(* PLC project tni_train, Dassault Systèmes ControlBuild 2019 FD01 Beta 2 *)
(* stored: creationDateTime 2018-09-11T17:45:24-01:00 *)

CONFIGURATION tni_train
  VAR_GLOBAL
    cab1/keyCabEnabled2 AT 97 : BOOL := false;
    cab1/keyCabDisabled2 AT 98 : BOOL := false;
    cab1/enableOpeningRightC1 AT 102 : BOOL := false;
    cab1/enableOpeningLeftC1 AT 104 : BOOL := false;
    cab1/enableClosingRightC1 AT 103 : BOOL := false;
    cab1/enableClosingLeftC1 AT 101 : BOOL := false;
    cab1/cabEnabled AT 99 : BOOL := false;
    cab1/cabDisabled AT 100 : BOOL := false;
    cab1/cabIncoherence AT 96 : BOOL := false;
    cab1/key2position/keyCabEnabled AT 109 : BOOL := false;
    cab1/key2position/keyCabDisabled AT 110 : BOOL := true;
    cab1/key2position/button AT 114 : BOOL := false;
    cab1/key2position/_X_10 AT 115 : BOOL := true;
    cab1/key2position/_X_11 AT 116 : BOOL := false;
    cab1/service_side/rightServiceSide AT 111 : BOOL := false;
    cab1/service_side/leftServiceSide AT 112 : BOOL := true;
    cab1/service_side/button AT 119 : BOOL := false;
    cab1/service_side/_X_10 AT 120 : BOOL := true;
    cab1/service_side/_X_11 AT 121 : BOOL := false;
    cab1/closingPB/PB AT 113 : BOOL := false;
    cab1/closingPB/button AT 124 : BOOL := false;
    cab1/closingPB/_X_10 AT 125 : BOOL := true;
    cab1/closingPB/_X_11 AT 126 : BOOL := false;
    cab1/trainSpeed/speed AT 17 : REAL := 0.0;
    cab1/cabControlPart/keyCabEnabled AT 109 : BOOL := false;
    cab1/cabControlPart/keyCabDisabled AT 110 : BOOL := true;
    cab1/cabControlPart/rightServiceSide AT 111 : BOOL := false;
    cab1/cabControlPart/leftServiceSide AT 112 : BOOL := true;
    cab1/cabControlPart/pbDoorClosing AT 113 : BOOL := false;
    cab1/cabControlPart/speed AT 17 : REAL := 0.0;
    cab1/cabControlPart/keyCabEnabled2 AT 97 : BOOL := false;
    cab1/cabControlPart/keyCabDisabled2 AT 98 : BOOL := false;
    cab1/cabControlPart/enableOpeningRightC1 AT 102 : BOOL := false;
    cab1/cabControlPart/enableOpeningLeftC1 AT 104 : BOOL := false;
    cab1/cabControlPart/enableClosingRightC1 AT 103 : BOOL := false;
    cab1/cabControlPart/enableClosingLeftC1 AT 101 : BOOL := false;
    cab1/cabControlPart/cabEnabled AT 99 : BOOL := false;
    cab1/cabControlPart/cabDisabled AT 100 : BOOL := false;
    cab1/cabControlPart/cabIncoherence AT 96 : BOOL := false;
    cab1/cabControlPart/limitLowSpeed AT 18 : REAL := 6.0;
    cab2/keyCabEnabled2 AT 99 : BOOL := false;
    cab2/keyCabDisabled2 AT 100 : BOOL := false;
    cab2/enableOpeningRightC1 AT 106 : BOOL := false;
    cab2/enableOpeningLeftC1 AT 108 : BOOL := false;
    cab2/enableClosingRightC1 AT 107 : BOOL := false;
    cab2/enableClosingLeftC1 AT 105 : BOOL := false;
    cab2/cabEnabled AT 97 : BOOL := false;
    cab2/cabDisabled AT 98 : BOOL := false;
    cab2/cabIncoherence AT 95 : BOOL := false;
    cab2/key2position/keyCabEnabled AT 129 : BOOL := false;
    cab2/key2position/keyCabDisabled AT 130 : BOOL := true;
    cab2/key2position/button AT 134 : BOOL := false;
    cab2/key2position/_X_10 AT 135 : BOOL := true;
    cab2/key2position/_X_11 AT 136 : BOOL := false;
    cab2/service_side/rightServiceSide AT 131 : BOOL := false;
    cab2/service_side/leftServiceSide AT 132 : BOOL := true;
    cab2/service_side/button AT 139 : BOOL := false;
    cab2/service_side/_X_10 AT 140 : BOOL := true;
    cab2/service_side/_X_11 AT 141 : BOOL := false;
    cab2/closingPB/PB AT 133 : BOOL := false;
    cab2/closingPB/button AT 144 : BOOL := false;
    cab2/closingPB/_X_10 AT 145 : BOOL := true;
    cab2/closingPB/_X_11 AT 146 : BOOL := false;
    cab2/trainSpeed/speed AT 19 : REAL := 0.0;
    cab2/cabControlPart/keyCabEnabled AT 129 : BOOL := false;
    cab2/cabControlPart/keyCabDisabled AT 130 : BOOL := true;
    cab2/cabControlPart/rightServiceSide AT 131 : BOOL := false;
    cab2/cabControlPart/leftServiceSide AT 132 : BOOL := true;
    cab2/cabControlPart/pbDoorClosing AT 133 : BOOL := false;
    cab2/cabControlPart/speed AT 19 : REAL := 0.0;
    cab2/cabControlPart/keyCabEnabled2 AT 99 : BOOL := false;
    cab2/cabControlPart/keyCabDisabled2 AT 100 : BOOL := false;
    cab2/cabControlPart/enableOpeningRightC1 AT 106 : BOOL := false;
    cab2/cabControlPart/enableOpeningLeftC1 AT 108 : BOOL := false;
    cab2/cabControlPart/enableClosingRightC1 AT 107 : BOOL := false;
    cab2/cabControlPart/enableClosingLeftC1 AT 105 : BOOL := false;
    cab2/cabControlPart/cabEnabled AT 97 : BOOL := false;
    cab2/cabControlPart/cabDisabled AT 98 : BOOL := false;
    cab2/cabControlPart/cabIncoherence AT 95 : BOOL := false;
    cab2/cabControlPart/limitLowSpeed AT 20 : REAL := 6.0;
    motorCar1/AuthorizationClosingLeftC1 AT 101 : BOOL := false;
    motorCar1/AuthorizationOpeningRightC1 AT 102 : BOOL := false;
    motorCar1/AuthorizationClosingRightC1 AT 103 : BOOL := false;
    motorCar1/AuthorizationOpeningLeftC1 AT 104 : BOOL := false;
    motorCar1/AuthorizationClosingLeftC2 AT 105 : BOOL := false;
    motorCar1/AuthorizationOpeningRightC2 AT 106 : BOOL := false;
    motorCar1/AuthorizationClosingRightC2 AT 107 : BOOL := false;
    motorCar1/AuthorizationOpeningLeftC2 AT 108 : BOOL := false;
    motorCar1/doorL1Closed AT 94 : BOOL := false;
    motorCar1/doorL1Opened AT 93 : BOOL := false;
    motorCar1/doorL1Fault AT 552 : DINT := 0;
    motorCar1/doorL2Closed AT 92 : BOOL := false;
    motorCar1/doorL2Opened AT 91 : BOOL := false;
    motorCar1/doorL2Fault AT 551 : DINT := 0;
    motorCar1/doorL3Closed AT 90 : BOOL := false;
    motorCar1/doorL3Opened AT 89 : BOOL := false;
    motorCar1/doorL3Fault AT 550 : DINT := 0;
    motorCar1/doorR1Closed AT 88 : BOOL := false;
    motorCar1/doorR1Opened AT 87 : BOOL := false;
    motorCar1/doorR1Fault AT 549 : DINT := 0;
    motorCar1/doorR2Closed AT 86 : BOOL := false;
    motorCar1/doorR2Opened AT 85 : BOOL := false;
    motorCar1/doorR2Fault AT 548 : DINT := 0;
    motorCar1/doorR3Closed AT 84 : BOOL := false;
    motorCar1/doorR3Opened AT 83 : BOOL := false;
    motorCar1/doorR3Fault AT 547 : DINT := 0;
    motorCar1/AlarmD1L AT 82 : BOOL := false;
    motorCar1/AlarmD2L AT 81 : BOOL := false;
    motorCar1/AlarmD3L AT 80 : BOOL := false;
    motorCar1/AlarmD1R AT 79 : BOOL := false;
    motorCar1/AlarmD2R AT 78 : BOOL := false;
    motorCar1/AlarmD3R AT 77 : BOOL := false;
    motorCar1/authorizations/AuthorizationClosingLeftC1 AT 101 : BOOL := false;
    motorCar1/authorizations/AuthorizationOpeningRightC1 AT 102 : BOOL := false;
    motorCar1/authorizations/AuthorizationClosingRightC1 AT 103 : BOOL := false;
    motorCar1/authorizations/AuthorizationOpeningLeftC1 AT 104 : BOOL := false;
    motorCar1/authorizations/AuthorizationClosingLeftC2 AT 105 : BOOL := false;
    motorCar1/authorizations/AuthorizationOpeningRightC2 AT 106 : BOOL := false;
    motorCar1/authorizations/AuthorizationClosingRightC2 AT 107 : BOOL := false;
    motorCar1/authorizations/AuthorizationOpeningLeftC2 AT 108 : BOOL := false;
    motorCar1/authorizations/AuthorizationOpeningLeft AT 161 : BOOL := false;
    motorCar1/authorizations/AuthorizationClosingLeft AT 162 : BOOL := false;
    motorCar1/authorizations/AuthorizationOpeningRight AT 163 : BOOL := false;
    motorCar1/authorizations/AuthorizationClosingRight AT 164 : BOOL := false;
    motorCar1/alarms/AlarmD1L AT 82 : BOOL := false;
    motorCar1/alarms/AlarmD2L AT 81 : BOOL := false;
    motorCar1/alarms/AlarmD3L AT 80 : BOOL := false;
    motorCar1/alarms/AlarmD1R AT 79 : BOOL := false;
    motorCar1/alarms/AlarmD2R AT 78 : BOOL := false;
    motorCar1/alarms/AlarmD3R AT 77 : BOOL := false;
    motorCar1/alarms/AlarmD1L/enableAlarm AT 176 : BOOL := false;
    motorCar1/alarms/AlarmD1L/resetKey AT 175 : BOOL := false;
    motorCar1/alarms/AlarmD1L/alarm AT 82 : BOOL := false;
    motorCar1/alarms/AlarmD1L/i_rs1 AT 553 : DINT := 0;
    motorCar1/alarms/AlarmD2L/enableAlarm AT 174 : BOOL := false;
    motorCar1/alarms/AlarmD2L/resetKey AT 173 : BOOL := false;
    motorCar1/alarms/AlarmD2L/alarm AT 81 : BOOL := false;
    motorCar1/alarms/AlarmD2L/i_rs1 AT 555 : DINT := 0;
    motorCar1/alarms/AlarmD3L/enableAlarm AT 172 : BOOL := false;
    motorCar1/alarms/AlarmD3L/resetKey AT 171 : BOOL := false;
    motorCar1/alarms/AlarmD3L/alarm AT 80 : BOOL := false;
    motorCar1/alarms/AlarmD3L/i_rs1 AT 557 : DINT := 0;
    motorCar1/alarms/AlarmD1R/enableAlarm AT 170 : BOOL := false;
    motorCar1/alarms/AlarmD1R/resetKey AT 169 : BOOL := false;
    motorCar1/alarms/AlarmD1R/alarm AT 79 : BOOL := false;
    motorCar1/alarms/AlarmD1R/i_rs1 AT 559 : DINT := 0;
    motorCar1/alarms/AlarmD2R/enableAlarm AT 168 : BOOL := false;
    motorCar1/alarms/AlarmD2R/resetKey AT 167 : BOOL := false;
    motorCar1/alarms/AlarmD2R/alarm AT 78 : BOOL := false;
    motorCar1/alarms/AlarmD2R/i_rs1 AT 561 : DINT := 0;
    motorCar1/alarms/AlarmD3R/enableAlarm AT 166 : BOOL := false;
    motorCar1/alarms/AlarmD3R/resetKey AT 165 : BOOL := false;
    motorCar1/alarms/AlarmD3R/alarm AT 77 : BOOL := false;
    motorCar1/alarms/AlarmD3R/i_rs1 AT 563 : DINT := 0;
    motorCar1/doorL1/compressedAir AT 26 : REAL := 200.0;
    motorCar1/doorL1/cmdSupply AT 160 : BOOL := true;
    motorCar1/doorL1/sensorSupply AT 159 : BOOL := true;
    motorCar1/doorL1/enableOpening AT 161 : BOOL := false;
    motorCar1/doorL1/enableClosing AT 162 : BOOL := false;
    motorCar1/doorL1/closedDoorState AT 94 : BOOL := false;
    motorCar1/doorL1/openedDoorState AT 93 : BOOL := false;
    motorCar1/doorL1/faultState AT 552 : DINT := 0;
    motorCar1/doorL1/doorPB/doorPB AT 189 : BOOL := false;
    motorCar1/doorL1/doorPB/button AT 193 : BOOL := false;
    motorCar1/doorL1/doorPB/_X_10 AT 194 : BOOL := true;
    motorCar1/doorL1/doorPB/_X_11 AT 195 : BOOL := false;
    motorCar1/doorL1/doorPB/_X_12 AT 196 : BOOL := false;
    motorCar1/doorL1/doorLocking/lockingCmd AT 183 : BOOL := false;
    motorCar1/doorL1/doorLocking/unlockingCmd AT 184 : BOOL := false;
    motorCar1/doorL1/doorLocking/doorLocked AT 187 : BOOL := false;
    motorCar1/doorL1/doorLocking/doorUnlocked AT 188 : BOOL := false;
    motorCar1/doorL1/doorLocking/lockActive AT 192 : BOOL := false;
    motorCar1/doorL1/doorLocking/i_rs1 AT 566 : DINT := 0;
    motorCar1/doorL1/doorLocking/d_unlockedSensor AT 198 : BOOL := false;
    motorCar1/doorL1/doorLocking/v_d_unlockedSensor AT 199 : BOOL := false;
    motorCar1/doorL1/doorLocking/d_lockedSensor AT 200 : BOOL := false;
    motorCar1/doorL1/doorLocking/v_d_lockedSensor AT 201 : BOOL := false;
    motorCar1/doorL1/doorControlPart/enableOpening AT 161 : BOOL := false;
    motorCar1/doorL1/doorControlPart/enableClosing AT 162 : BOOL := false;
    motorCar1/doorL1/doorControlPart/openedDoor AT 185 : BOOL := false;
    motorCar1/doorL1/doorControlPart/closedDoor AT 186 : BOOL := false;
    motorCar1/doorL1/doorControlPart/lockedDoor AT 187 : BOOL := false;
    motorCar1/doorL1/doorControlPart/unlockedDoor AT 188 : BOOL := false;
    motorCar1/doorL1/doorControlPart/openingRequest AT 189 : BOOL := false;
    motorCar1/doorL1/doorControlPart/doorOpeningCmd AT 190 : BOOL := false;
    motorCar1/doorL1/doorControlPart/doorClosingCmd AT 191 : BOOL := false;
    motorCar1/doorL1/doorControlPart/doorLockingCmd AT 183 : BOOL := false;
    motorCar1/doorL1/doorControlPart/doorUnlockingCmd AT 184 : BOOL := false;
    motorCar1/doorL1/doorControlPart/closedDoorState AT 94 : BOOL := false;
    motorCar1/doorL1/doorControlPart/openedDoorState AT 93 : BOOL := false;
    motorCar1/doorL1/doorControlPart/faultState AT 552 : DINT := 0;
    motorCar1/doorL1/doorControlPart/_X_10 AT 203 : BOOL := true;
    motorCar1/doorL1/doorControlPart/_X_11 AT 204 : BOOL := false;
    motorCar1/doorL1/doorControlPart/_X_12 AT 205 : BOOL := false;
    motorCar1/doorL1/doorControlPart/_X_13 AT 206 : BOOL := false;
    motorCar1/doorL1/doorControlPart/_X_14 AT 207 : BOOL := false;
    motorCar1/doorL1/doorControlPart/_X_15 AT 208 : BOOL := false;
    motorCar1/doorL1/doorControlPart/_X_16 AT 209 : BOOL := false;
    motorCar1/doorL1/door/compressedAir AT 26 : REAL := 200.0;
    motorCar1/doorL1/door/cmdSupply AT 160 : BOOL := true;
    motorCar1/doorL1/door/sensorSupply AT 159 : BOOL := true;
    motorCar1/doorL1/door/openDoorCmd AT 190 : BOOL := false;
    motorCar1/doorL1/door/closeDoorCmd AT 191 : BOOL := false;
    motorCar1/doorL1/door/lockActive AT 192 : BOOL := false;
    motorCar1/doorL1/door/doorOpened AT 185 : BOOL := false;
    motorCar1/doorL1/door/doorClosed AT 186 : BOOL := false;
    motorCar1/doorL1/door/increment AT 27 : REAL := 0.0;
    motorCar1/doorL1/door/openDoor AT 216 : BOOL := false;
    motorCar1/doorL1/door/closeDoor AT 217 : BOOL := false;
    motorCar1/doorL1/door/doorPosition AT 28 : REAL := 0.0;
    motorCar1/doorL1/door/length AT 29 : REAL := 1000.0;
    motorCar1/doorL1/door/doorClosedSensorLogic AT 218 : BOOL := true;
    motorCar1/doorL1/door/doorOpenedSensorLogic AT 219 : BOOL := true;
    motorCar1/doorL1/door/d_locking AT 220 : BOOL := false;
    motorCar1/doorL1/door/v_d_locking AT 30 : REAL := 50.0;
    motorCar1/doorL1/door/d_doorClosedSensor AT 221 : BOOL := false;
    motorCar1/doorL1/door/v_d_doorClosedSensor AT 222 : BOOL := false;
    motorCar1/doorL1/door/d_doorOpenedSensor AT 223 : BOOL := false;
    motorCar1/doorL1/door/v_d_doorOpenedSensor AT 224 : BOOL := false;
    motorCar1/doorL2/compressedAir AT 25 : REAL := 200.0;
    motorCar1/doorL2/cmdSupply AT 158 : BOOL := true;
    motorCar1/doorL2/sensorSupply AT 157 : BOOL := true;
    motorCar1/doorL2/enableOpening AT 161 : BOOL := false;
    motorCar1/doorL2/enableClosing AT 162 : BOOL := false;
    motorCar1/doorL2/closedDoorState AT 92 : BOOL := false;
    motorCar1/doorL2/openedDoorState AT 91 : BOOL := false;
    motorCar1/doorL2/faultState AT 551 : DINT := 0;
    motorCar1/doorL2/doorPB/doorPB AT 231 : BOOL := false;
    motorCar1/doorL2/doorPB/button AT 235 : BOOL := false;
    motorCar1/doorL2/doorPB/_X_10 AT 236 : BOOL := true;
    motorCar1/doorL2/doorPB/_X_11 AT 237 : BOOL := false;
    motorCar1/doorL2/doorPB/_X_12 AT 238 : BOOL := false;
    motorCar1/doorL2/doorLocking/lockingCmd AT 225 : BOOL := false;
    motorCar1/doorL2/doorLocking/unlockingCmd AT 226 : BOOL := false;
    motorCar1/doorL2/doorLocking/doorLocked AT 229 : BOOL := false;
    motorCar1/doorL2/doorLocking/doorUnlocked AT 230 : BOOL := false;
    motorCar1/doorL2/doorLocking/lockActive AT 234 : BOOL := false;
    motorCar1/doorL2/doorLocking/i_rs1 AT 569 : DINT := 0;
    motorCar1/doorL2/doorLocking/d_unlockedSensor AT 240 : BOOL := false;
    motorCar1/doorL2/doorLocking/v_d_unlockedSensor AT 241 : BOOL := false;
    motorCar1/doorL2/doorLocking/d_lockedSensor AT 242 : BOOL := false;
    motorCar1/doorL2/doorLocking/v_d_lockedSensor AT 243 : BOOL := false;
    motorCar1/doorL2/doorControlPart/enableOpening AT 161 : BOOL := false;
    motorCar1/doorL2/doorControlPart/enableClosing AT 162 : BOOL := false;
    motorCar1/doorL2/doorControlPart/openedDoor AT 227 : BOOL := false;
    motorCar1/doorL2/doorControlPart/closedDoor AT 228 : BOOL := false;
    motorCar1/doorL2/doorControlPart/lockedDoor AT 229 : BOOL := false;
    motorCar1/doorL2/doorControlPart/unlockedDoor AT 230 : BOOL := false;
    motorCar1/doorL2/doorControlPart/openingRequest AT 231 : BOOL := false;
    motorCar1/doorL2/doorControlPart/doorOpeningCmd AT 232 : BOOL := false;
    motorCar1/doorL2/doorControlPart/doorClosingCmd AT 233 : BOOL := false;
    motorCar1/doorL2/doorControlPart/doorLockingCmd AT 225 : BOOL := false;
    motorCar1/doorL2/doorControlPart/doorUnlockingCmd AT 226 : BOOL := false;
    motorCar1/doorL2/doorControlPart/closedDoorState AT 92 : BOOL := false;
    motorCar1/doorL2/doorControlPart/openedDoorState AT 91 : BOOL := false;
    motorCar1/doorL2/doorControlPart/faultState AT 551 : DINT := 0;
    motorCar1/doorL2/doorControlPart/_X_10 AT 245 : BOOL := true;
    motorCar1/doorL2/doorControlPart/_X_11 AT 246 : BOOL := false;
    motorCar1/doorL2/doorControlPart/_X_12 AT 247 : BOOL := false;
    motorCar1/doorL2/doorControlPart/_X_13 AT 248 : BOOL := false;
    motorCar1/doorL2/doorControlPart/_X_14 AT 249 : BOOL := false;
    motorCar1/doorL2/doorControlPart/_X_15 AT 250 : BOOL := false;
    motorCar1/doorL2/doorControlPart/_X_16 AT 251 : BOOL := false;
    motorCar1/doorL2/door/compressedAir AT 25 : REAL := 200.0;
    motorCar1/doorL2/door/cmdSupply AT 158 : BOOL := true;
    motorCar1/doorL2/door/sensorSupply AT 157 : BOOL := true;
    motorCar1/doorL2/door/openDoorCmd AT 232 : BOOL := false;
    motorCar1/doorL2/door/closeDoorCmd AT 233 : BOOL := false;
    motorCar1/doorL2/door/lockActive AT 234 : BOOL := false;
    motorCar1/doorL2/door/doorOpened AT 227 : BOOL := false;
    motorCar1/doorL2/door/doorClosed AT 228 : BOOL := false;
    motorCar1/doorL2/door/increment AT 31 : REAL := 0.0;
    motorCar1/doorL2/door/openDoor AT 258 : BOOL := false;
    motorCar1/doorL2/door/closeDoor AT 259 : BOOL := false;
    motorCar1/doorL2/door/doorPosition AT 32 : REAL := 0.0;
    motorCar1/doorL2/door/length AT 33 : REAL := 1000.0;
    motorCar1/doorL2/door/doorClosedSensorLogic AT 260 : BOOL := true;
    motorCar1/doorL2/door/doorOpenedSensorLogic AT 261 : BOOL := true;
    motorCar1/doorL2/door/d_locking AT 262 : BOOL := false;
    motorCar1/doorL2/door/v_d_locking AT 34 : REAL := 50.0;
    motorCar1/doorL2/door/d_doorClosedSensor AT 263 : BOOL := false;
    motorCar1/doorL2/door/v_d_doorClosedSensor AT 264 : BOOL := false;
    motorCar1/doorL2/door/d_doorOpenedSensor AT 265 : BOOL := false;
    motorCar1/doorL2/door/v_d_doorOpenedSensor AT 266 : BOOL := false;
    motorCar1/doorL3/compressedAir AT 24 : REAL := 200.0;
    motorCar1/doorL3/cmdSupply AT 156 : BOOL := true;
    motorCar1/doorL3/sensorSupply AT 155 : BOOL := true;
    motorCar1/doorL3/enableOpening AT 161 : BOOL := false;
    motorCar1/doorL3/enableClosing AT 162 : BOOL := false;
    motorCar1/doorL3/closedDoorState AT 90 : BOOL := false;
    motorCar1/doorL3/openedDoorState AT 89 : BOOL := false;
    motorCar1/doorL3/faultState AT 550 : DINT := 0;
    motorCar1/doorL3/doorPB/doorPB AT 273 : BOOL := false;
    motorCar1/doorL3/doorPB/button AT 277 : BOOL := false;
    motorCar1/doorL3/doorPB/_X_10 AT 278 : BOOL := true;
    motorCar1/doorL3/doorPB/_X_11 AT 279 : BOOL := false;
    motorCar1/doorL3/doorPB/_X_12 AT 280 : BOOL := false;
    motorCar1/doorL3/doorLocking/lockingCmd AT 267 : BOOL := false;
    motorCar1/doorL3/doorLocking/unlockingCmd AT 268 : BOOL := false;
    motorCar1/doorL3/doorLocking/doorLocked AT 271 : BOOL := false;
    motorCar1/doorL3/doorLocking/doorUnlocked AT 272 : BOOL := false;
    motorCar1/doorL3/doorLocking/lockActive AT 276 : BOOL := false;
    motorCar1/doorL3/doorLocking/i_rs1 AT 572 : DINT := 0;
    motorCar1/doorL3/doorLocking/d_unlockedSensor AT 282 : BOOL := false;
    motorCar1/doorL3/doorLocking/v_d_unlockedSensor AT 283 : BOOL := false;
    motorCar1/doorL3/doorLocking/d_lockedSensor AT 284 : BOOL := false;
    motorCar1/doorL3/doorLocking/v_d_lockedSensor AT 285 : BOOL := false;
    motorCar1/doorL3/doorControlPart/enableOpening AT 161 : BOOL := false;
    motorCar1/doorL3/doorControlPart/enableClosing AT 162 : BOOL := false;
    motorCar1/doorL3/doorControlPart/openedDoor AT 269 : BOOL := false;
    motorCar1/doorL3/doorControlPart/closedDoor AT 270 : BOOL := false;
    motorCar1/doorL3/doorControlPart/lockedDoor AT 271 : BOOL := false;
    motorCar1/doorL3/doorControlPart/unlockedDoor AT 272 : BOOL := false;
    motorCar1/doorL3/doorControlPart/openingRequest AT 273 : BOOL := false;
    motorCar1/doorL3/doorControlPart/doorOpeningCmd AT 274 : BOOL := false;
    motorCar1/doorL3/doorControlPart/doorClosingCmd AT 275 : BOOL := false;
    motorCar1/doorL3/doorControlPart/doorLockingCmd AT 267 : BOOL := false;
    motorCar1/doorL3/doorControlPart/doorUnlockingCmd AT 268 : BOOL := false;
    motorCar1/doorL3/doorControlPart/closedDoorState AT 90 : BOOL := false;
    motorCar1/doorL3/doorControlPart/openedDoorState AT 89 : BOOL := false;
    motorCar1/doorL3/doorControlPart/faultState AT 550 : DINT := 0;
    motorCar1/doorL3/doorControlPart/_X_10 AT 287 : BOOL := true;
    motorCar1/doorL3/doorControlPart/_X_11 AT 288 : BOOL := false;
    motorCar1/doorL3/doorControlPart/_X_12 AT 289 : BOOL := false;
    motorCar1/doorL3/doorControlPart/_X_13 AT 290 : BOOL := false;
    motorCar1/doorL3/doorControlPart/_X_14 AT 291 : BOOL := false;
    motorCar1/doorL3/doorControlPart/_X_15 AT 292 : BOOL := false;
    motorCar1/doorL3/doorControlPart/_X_16 AT 293 : BOOL := false;
    motorCar1/doorL3/door/compressedAir AT 24 : REAL := 200.0;
    motorCar1/doorL3/door/cmdSupply AT 156 : BOOL := true;
    motorCar1/doorL3/door/sensorSupply AT 155 : BOOL := true;
    motorCar1/doorL3/door/openDoorCmd AT 274 : BOOL := false;
    motorCar1/doorL3/door/closeDoorCmd AT 275 : BOOL := false;
    motorCar1/doorL3/door/lockActive AT 276 : BOOL := false;
    motorCar1/doorL3/door/doorOpened AT 269 : BOOL := false;
    motorCar1/doorL3/door/doorClosed AT 270 : BOOL := false;
    motorCar1/doorL3/door/increment AT 35 : REAL := 0.0;
    motorCar1/doorL3/door/openDoor AT 300 : BOOL := false;
    motorCar1/doorL3/door/closeDoor AT 301 : BOOL := false;
    motorCar1/doorL3/door/doorPosition AT 36 : REAL := 0.0;
    motorCar1/doorL3/door/length AT 37 : REAL := 1000.0;
    motorCar1/doorL3/door/doorClosedSensorLogic AT 302 : BOOL := true;
    motorCar1/doorL3/door/doorOpenedSensorLogic AT 303 : BOOL := true;
    motorCar1/doorL3/door/d_locking AT 304 : BOOL := false;
    motorCar1/doorL3/door/v_d_locking AT 38 : REAL := 50.0;
    motorCar1/doorL3/door/d_doorClosedSensor AT 305 : BOOL := false;
    motorCar1/doorL3/door/v_d_doorClosedSensor AT 306 : BOOL := false;
    motorCar1/doorL3/door/d_doorOpenedSensor AT 307 : BOOL := false;
    motorCar1/doorL3/door/v_d_doorOpenedSensor AT 308 : BOOL := false;
    motorCar1/doorR1/compressedAir AT 23 : REAL := 200.0;
    motorCar1/doorR1/cmdSupply AT 154 : BOOL := true;
    motorCar1/doorR1/sensorSupply AT 153 : BOOL := true;
    motorCar1/doorR1/enableOpening AT 163 : BOOL := false;
    motorCar1/doorR1/enableClosing AT 164 : BOOL := false;
    motorCar1/doorR1/closedDoorState AT 88 : BOOL := false;
    motorCar1/doorR1/openedDoorState AT 87 : BOOL := false;
    motorCar1/doorR1/faultState AT 549 : DINT := 0;
    motorCar1/doorR1/doorPB/doorPB AT 315 : BOOL := false;
    motorCar1/doorR1/doorPB/button AT 319 : BOOL := false;
    motorCar1/doorR1/doorPB/_X_10 AT 320 : BOOL := true;
    motorCar1/doorR1/doorPB/_X_11 AT 321 : BOOL := false;
    motorCar1/doorR1/doorPB/_X_12 AT 322 : BOOL := false;
    motorCar1/doorR1/doorLocking/lockingCmd AT 309 : BOOL := false;
    motorCar1/doorR1/doorLocking/unlockingCmd AT 310 : BOOL := false;
    motorCar1/doorR1/doorLocking/doorLocked AT 313 : BOOL := false;
    motorCar1/doorR1/doorLocking/doorUnlocked AT 314 : BOOL := false;
    motorCar1/doorR1/doorLocking/lockActive AT 318 : BOOL := false;
    motorCar1/doorR1/doorLocking/i_rs1 AT 575 : DINT := 0;
    motorCar1/doorR1/doorLocking/d_unlockedSensor AT 324 : BOOL := false;
    motorCar1/doorR1/doorLocking/v_d_unlockedSensor AT 325 : BOOL := false;
    motorCar1/doorR1/doorLocking/d_lockedSensor AT 326 : BOOL := false;
    motorCar1/doorR1/doorLocking/v_d_lockedSensor AT 327 : BOOL := false;
    motorCar1/doorR1/doorControlPart/enableOpening AT 163 : BOOL := false;
    motorCar1/doorR1/doorControlPart/enableClosing AT 164 : BOOL := false;
    motorCar1/doorR1/doorControlPart/openedDoor AT 311 : BOOL := false;
    motorCar1/doorR1/doorControlPart/closedDoor AT 312 : BOOL := false;
    motorCar1/doorR1/doorControlPart/lockedDoor AT 313 : BOOL := false;
    motorCar1/doorR1/doorControlPart/unlockedDoor AT 314 : BOOL := false;
    motorCar1/doorR1/doorControlPart/openingRequest AT 315 : BOOL := false;
    motorCar1/doorR1/doorControlPart/doorOpeningCmd AT 316 : BOOL := false;
    motorCar1/doorR1/doorControlPart/doorClosingCmd AT 317 : BOOL := false;
    motorCar1/doorR1/doorControlPart/doorLockingCmd AT 309 : BOOL := false;
    motorCar1/doorR1/doorControlPart/doorUnlockingCmd AT 310 : BOOL := false;
    motorCar1/doorR1/doorControlPart/closedDoorState AT 88 : BOOL := false;
    motorCar1/doorR1/doorControlPart/openedDoorState AT 87 : BOOL := false;
    motorCar1/doorR1/doorControlPart/faultState AT 549 : DINT := 0;
    motorCar1/doorR1/doorControlPart/_X_10 AT 329 : BOOL := true;
    motorCar1/doorR1/doorControlPart/_X_11 AT 330 : BOOL := false;
    motorCar1/doorR1/doorControlPart/_X_12 AT 331 : BOOL := false;
    motorCar1/doorR1/doorControlPart/_X_13 AT 332 : BOOL := false;
    motorCar1/doorR1/doorControlPart/_X_14 AT 333 : BOOL := false;
    motorCar1/doorR1/doorControlPart/_X_15 AT 334 : BOOL := false;
    motorCar1/doorR1/doorControlPart/_X_16 AT 335 : BOOL := false;
    motorCar1/doorR1/door/compressedAir AT 23 : REAL := 200.0;
    motorCar1/doorR1/door/cmdSupply AT 154 : BOOL := true;
    motorCar1/doorR1/door/sensorSupply AT 153 : BOOL := true;
    motorCar1/doorR1/door/openDoorCmd AT 316 : BOOL := false;
    motorCar1/doorR1/door/closeDoorCmd AT 317 : BOOL := false;
    motorCar1/doorR1/door/lockActive AT 318 : BOOL := false;
    motorCar1/doorR1/door/doorOpened AT 311 : BOOL := false;
    motorCar1/doorR1/door/doorClosed AT 312 : BOOL := false;
    motorCar1/doorR1/door/increment AT 39 : REAL := 0.0;
    motorCar1/doorR1/door/openDoor AT 342 : BOOL := false;
    motorCar1/doorR1/door/closeDoor AT 343 : BOOL := false;
    motorCar1/doorR1/door/doorPosition AT 40 : REAL := 0.0;
    motorCar1/doorR1/door/length AT 41 : REAL := 1000.0;
    motorCar1/doorR1/door/doorClosedSensorLogic AT 344 : BOOL := true;
    motorCar1/doorR1/door/doorOpenedSensorLogic AT 345 : BOOL := true;
    motorCar1/doorR1/door/d_locking AT 346 : BOOL := false;
    motorCar1/doorR1/door/v_d_locking AT 42 : REAL := 50.0;
    motorCar1/doorR1/door/d_doorClosedSensor AT 347 : BOOL := false;
    motorCar1/doorR1/door/v_d_doorClosedSensor AT 348 : BOOL := false;
    motorCar1/doorR1/door/d_doorOpenedSensor AT 349 : BOOL := false;
    motorCar1/doorR1/door/v_d_doorOpenedSensor AT 350 : BOOL := false;
    motorCar1/doorR2/compressedAir AT 22 : REAL := 200.0;
    motorCar1/doorR2/cmdSupply AT 152 : BOOL := true;
    motorCar1/doorR2/sensorSupply AT 151 : BOOL := true;
    motorCar1/doorR2/enableOpening AT 163 : BOOL := false;
    motorCar1/doorR2/enableClosing AT 164 : BOOL := false;
    motorCar1/doorR2/closedDoorState AT 86 : BOOL := false;
    motorCar1/doorR2/openedDoorState AT 85 : BOOL := false;
    motorCar1/doorR2/faultState AT 548 : DINT := 0;
    motorCar1/doorR2/doorPB/doorPB AT 357 : BOOL := false;
    motorCar1/doorR2/doorPB/button AT 361 : BOOL := false;
    motorCar1/doorR2/doorPB/_X_10 AT 362 : BOOL := true;
    motorCar1/doorR2/doorPB/_X_11 AT 363 : BOOL := false;
    motorCar1/doorR2/doorPB/_X_12 AT 364 : BOOL := false;
    motorCar1/doorR2/doorLocking/lockingCmd AT 351 : BOOL := false;
    motorCar1/doorR2/doorLocking/unlockingCmd AT 352 : BOOL := false;
    motorCar1/doorR2/doorLocking/doorLocked AT 355 : BOOL := false;
    motorCar1/doorR2/doorLocking/doorUnlocked AT 356 : BOOL := false;
    motorCar1/doorR2/doorLocking/lockActive AT 360 : BOOL := false;
    motorCar1/doorR2/doorLocking/i_rs1 AT 578 : DINT := 0;
    motorCar1/doorR2/doorLocking/d_unlockedSensor AT 366 : BOOL := false;
    motorCar1/doorR2/doorLocking/v_d_unlockedSensor AT 367 : BOOL := false;
    motorCar1/doorR2/doorLocking/d_lockedSensor AT 368 : BOOL := false;
    motorCar1/doorR2/doorLocking/v_d_lockedSensor AT 369 : BOOL := false;
    motorCar1/doorR2/doorControlPart/enableOpening AT 163 : BOOL := false;
    motorCar1/doorR2/doorControlPart/enableClosing AT 164 : BOOL := false;
    motorCar1/doorR2/doorControlPart/openedDoor AT 353 : BOOL := false;
    motorCar1/doorR2/doorControlPart/closedDoor AT 354 : BOOL := false;
    motorCar1/doorR2/doorControlPart/lockedDoor AT 355 : BOOL := false;
    motorCar1/doorR2/doorControlPart/unlockedDoor AT 356 : BOOL := false;
    motorCar1/doorR2/doorControlPart/openingRequest AT 357 : BOOL := false;
    motorCar1/doorR2/doorControlPart/doorOpeningCmd AT 358 : BOOL := false;
    motorCar1/doorR2/doorControlPart/doorClosingCmd AT 359 : BOOL := false;
    motorCar1/doorR2/doorControlPart/doorLockingCmd AT 351 : BOOL := false;
    motorCar1/doorR2/doorControlPart/doorUnlockingCmd AT 352 : BOOL := false;
    motorCar1/doorR2/doorControlPart/closedDoorState AT 86 : BOOL := false;
    motorCar1/doorR2/doorControlPart/openedDoorState AT 85 : BOOL := false;
    motorCar1/doorR2/doorControlPart/faultState AT 548 : DINT := 0;
    motorCar1/doorR2/doorControlPart/_X_10 AT 371 : BOOL := true;
    motorCar1/doorR2/doorControlPart/_X_11 AT 372 : BOOL := false;
    motorCar1/doorR2/doorControlPart/_X_12 AT 373 : BOOL := false;
    motorCar1/doorR2/doorControlPart/_X_13 AT 374 : BOOL := false;
    motorCar1/doorR2/doorControlPart/_X_14 AT 375 : BOOL := false;
    motorCar1/doorR2/doorControlPart/_X_15 AT 376 : BOOL := false;
    motorCar1/doorR2/doorControlPart/_X_16 AT 377 : BOOL := false;
    motorCar1/doorR2/door/compressedAir AT 22 : REAL := 200.0;
    motorCar1/doorR2/door/cmdSupply AT 152 : BOOL := true;
    motorCar1/doorR2/door/sensorSupply AT 151 : BOOL := true;
    motorCar1/doorR2/door/openDoorCmd AT 358 : BOOL := false;
    motorCar1/doorR2/door/closeDoorCmd AT 359 : BOOL := false;
    motorCar1/doorR2/door/lockActive AT 360 : BOOL := false;
    motorCar1/doorR2/door/doorOpened AT 353 : BOOL := false;
    motorCar1/doorR2/door/doorClosed AT 354 : BOOL := false;
    motorCar1/doorR2/door/increment AT 43 : REAL := 0.0;
    motorCar1/doorR2/door/openDoor AT 384 : BOOL := false;
    motorCar1/doorR2/door/closeDoor AT 385 : BOOL := false;
    motorCar1/doorR2/door/doorPosition AT 44 : REAL := 0.0;
    motorCar1/doorR2/door/length AT 45 : REAL := 1000.0;
    motorCar1/doorR2/door/doorClosedSensorLogic AT 386 : BOOL := true;
    motorCar1/doorR2/door/doorOpenedSensorLogic AT 387 : BOOL := true;
    motorCar1/doorR2/door/d_locking AT 388 : BOOL := false;
    motorCar1/doorR2/door/v_d_locking AT 46 : REAL := 50.0;
    motorCar1/doorR2/door/d_doorClosedSensor AT 389 : BOOL := false;
    motorCar1/doorR2/door/v_d_doorClosedSensor AT 390 : BOOL := false;
    motorCar1/doorR2/door/d_doorOpenedSensor AT 391 : BOOL := false;
    motorCar1/doorR2/door/v_d_doorOpenedSensor AT 392 : BOOL := false;
    motorCar1/doorR3/compressedAir AT 21 : REAL := 200.0;
    motorCar1/doorR3/cmdSupply AT 150 : BOOL := true;
    motorCar1/doorR3/sensorSupply AT 149 : BOOL := true;
    motorCar1/doorR3/enableOpening AT 163 : BOOL := false;
    motorCar1/doorR3/enableClosing AT 164 : BOOL := false;
    motorCar1/doorR3/closedDoorState AT 84 : BOOL := false;
    motorCar1/doorR3/openedDoorState AT 83 : BOOL := false;
    motorCar1/doorR3/faultState AT 547 : DINT := 0;
    motorCar1/doorR3/doorPB/doorPB AT 399 : BOOL := false;
    motorCar1/doorR3/doorPB/button AT 403 : BOOL := false;
    motorCar1/doorR3/doorPB/_X_10 AT 404 : BOOL := true;
    motorCar1/doorR3/doorPB/_X_11 AT 405 : BOOL := false;
    motorCar1/doorR3/doorPB/_X_12 AT 406 : BOOL := false;
    motorCar1/doorR3/doorLocking/lockingCmd AT 393 : BOOL := false;
    motorCar1/doorR3/doorLocking/unlockingCmd AT 394 : BOOL := false;
    motorCar1/doorR3/doorLocking/doorLocked AT 397 : BOOL := false;
    motorCar1/doorR3/doorLocking/doorUnlocked AT 398 : BOOL := false;
    motorCar1/doorR3/doorLocking/lockActive AT 402 : BOOL := false;
    motorCar1/doorR3/doorLocking/i_rs1 AT 581 : DINT := 0;
    motorCar1/doorR3/doorLocking/d_unlockedSensor AT 408 : BOOL := false;
    motorCar1/doorR3/doorLocking/v_d_unlockedSensor AT 409 : BOOL := false;
    motorCar1/doorR3/doorLocking/d_lockedSensor AT 410 : BOOL := false;
    motorCar1/doorR3/doorLocking/v_d_lockedSensor AT 411 : BOOL := false;
    motorCar1/doorR3/doorControlPart/enableOpening AT 163 : BOOL := false;
    motorCar1/doorR3/doorControlPart/enableClosing AT 164 : BOOL := false;
    motorCar1/doorR3/doorControlPart/openedDoor AT 395 : BOOL := false;
    motorCar1/doorR3/doorControlPart/closedDoor AT 396 : BOOL := false;
    motorCar1/doorR3/doorControlPart/lockedDoor AT 397 : BOOL := false;
    motorCar1/doorR3/doorControlPart/unlockedDoor AT 398 : BOOL := false;
    motorCar1/doorR3/doorControlPart/openingRequest AT 399 : BOOL := false;
    motorCar1/doorR3/doorControlPart/doorOpeningCmd AT 400 : BOOL := false;
    motorCar1/doorR3/doorControlPart/doorClosingCmd AT 401 : BOOL := false;
    motorCar1/doorR3/doorControlPart/doorLockingCmd AT 393 : BOOL := false;
    motorCar1/doorR3/doorControlPart/doorUnlockingCmd AT 394 : BOOL := false;
    motorCar1/doorR3/doorControlPart/closedDoorState AT 84 : BOOL := false;
    motorCar1/doorR3/doorControlPart/openedDoorState AT 83 : BOOL := false;
    motorCar1/doorR3/doorControlPart/faultState AT 547 : DINT := 0;
    motorCar1/doorR3/doorControlPart/_X_10 AT 413 : BOOL := true;
    motorCar1/doorR3/doorControlPart/_X_11 AT 414 : BOOL := false;
    motorCar1/doorR3/doorControlPart/_X_12 AT 415 : BOOL := false;
    motorCar1/doorR3/doorControlPart/_X_13 AT 416 : BOOL := false;
    motorCar1/doorR3/doorControlPart/_X_14 AT 417 : BOOL := false;
    motorCar1/doorR3/doorControlPart/_X_15 AT 418 : BOOL := false;
    motorCar1/doorR3/doorControlPart/_X_16 AT 419 : BOOL := false;
    motorCar1/doorR3/door/compressedAir AT 21 : REAL := 200.0;
    motorCar1/doorR3/door/cmdSupply AT 150 : BOOL := true;
    motorCar1/doorR3/door/sensorSupply AT 149 : BOOL := true;
    motorCar1/doorR3/door/openDoorCmd AT 400 : BOOL := false;
    motorCar1/doorR3/door/closeDoorCmd AT 401 : BOOL := false;
    motorCar1/doorR3/door/lockActive AT 402 : BOOL := false;
    motorCar1/doorR3/door/doorOpened AT 395 : BOOL := false;
    motorCar1/doorR3/door/doorClosed AT 396 : BOOL := false;
    motorCar1/doorR3/door/increment AT 47 : REAL := 0.0;
    motorCar1/doorR3/door/openDoor AT 426 : BOOL := false;
    motorCar1/doorR3/door/closeDoor AT 427 : BOOL := false;
    motorCar1/doorR3/door/doorPosition AT 48 : REAL := 0.0;
    motorCar1/doorR3/door/length AT 49 : REAL := 1000.0;
    motorCar1/doorR3/door/doorClosedSensorLogic AT 428 : BOOL := true;
    motorCar1/doorR3/door/doorOpenedSensorLogic AT 429 : BOOL := true;
    motorCar1/doorR3/door/d_locking AT 430 : BOOL := false;
    motorCar1/doorR3/door/v_d_locking AT 50 : REAL := 50.0;
    motorCar1/doorR3/door/d_doorClosedSensor AT 431 : BOOL := false;
    motorCar1/doorR3/door/v_d_doorClosedSensor AT 432 : BOOL := false;
    motorCar1/doorR3/door/d_doorOpenedSensor AT 433 : BOOL := false;
    motorCar1/doorR3/door/v_d_doorOpenedSensor AT 434 : BOOL := false;
    car1/AuthorizationClosingLeftC1 AT 101 : BOOL := false;
    car1/AuthorizationOpeningRightC1 AT 102 : BOOL := false;
    car1/AuthorizationClosingRightC1 AT 103 : BOOL := false;
    car1/AuthorizationOpeningLeftC1 AT 104 : BOOL := false;
    car1/AuthorizationClosingLeftC2 AT 105 : BOOL := false;
    car1/AuthorizationOpeningRightC2 AT 106 : BOOL := false;
    car1/AuthorizationClosingRightC2 AT 107 : BOOL := false;
    car1/AuthorizationOpeningLeftC2 AT 108 : BOOL := false;
    car1/doorL1Closed AT 76 : BOOL := false;
    car1/doorL1Opened AT 75 : BOOL := false;
    car1/doorL1Fault AT 546 : DINT := 0;
    car1/doorL2Closed AT 74 : BOOL := false;
    car1/doorL2Opened AT 73 : BOOL := false;
    car1/doorL2Fault AT 545 : DINT := 0;
    car1/doorL3Closed AT 72 : BOOL := false;
    car1/doorL3Opened AT 71 : BOOL := false;
    car1/doorL3Fault AT 544 : DINT := 0;
    car1/doorR1Closed AT 70 : BOOL := false;
    car1/doorR1Opened AT 69 : BOOL := false;
    car1/doorR1Fault AT 543 : DINT := 0;
    car1/doorR2Closed AT 68 : BOOL := false;
    car1/doorR2Opened AT 67 : BOOL := false;
    car1/doorR2Fault AT 542 : DINT := 0;
    car1/doorR3Closed AT 66 : BOOL := false;
    car1/doorR3Opened AT 65 : BOOL := false;
    car1/doorR3Fault AT 541 : DINT := 0;
    car1/AlarmD1L AT 64 : BOOL := false;
    car1/AlarmD2L AT 63 : BOOL := false;
    car1/AlarmD3L AT 62 : BOOL := false;
    car1/AlarmD1R AT 61 : BOOL := false;
    car1/AlarmD2R AT 60 : BOOL := false;
    car1/AlarmD3R AT 59 : BOOL := false;
    car1/authorizations/AuthorizationClosingLeftC1 AT 101 : BOOL := false;
    car1/authorizations/AuthorizationOpeningRightC1 AT 102 : BOOL := false;
    car1/authorizations/AuthorizationClosingRightC1 AT 103 : BOOL := false;
    car1/authorizations/AuthorizationOpeningLeftC1 AT 104 : BOOL := false;
    car1/authorizations/AuthorizationClosingLeftC2 AT 105 : BOOL := false;
    car1/authorizations/AuthorizationOpeningRightC2 AT 106 : BOOL := false;
    car1/authorizations/AuthorizationClosingRightC2 AT 107 : BOOL := false;
    car1/authorizations/AuthorizationOpeningLeftC2 AT 108 : BOOL := false;
    car1/authorizations/AuthorizationOpeningLeft AT 447 : BOOL := false;
    car1/authorizations/AuthorizationClosingLeft AT 448 : BOOL := false;
    car1/authorizations/AuthorizationOpeningRight AT 449 : BOOL := false;
    car1/authorizations/AuthorizationClosingRight AT 450 : BOOL := false;
    car1/alarms/AlarmD1L AT 64 : BOOL := false;
    car1/alarms/AlarmD2L AT 63 : BOOL := false;
    car1/alarms/AlarmD3L AT 62 : BOOL := false;
    car1/alarms/AlarmD1R AT 61 : BOOL := false;
    car1/alarms/AlarmD2R AT 60 : BOOL := false;
    car1/alarms/AlarmD3R AT 59 : BOOL := false;
    car1/alarms/AlarmD1L/enableAlarm AT 462 : BOOL := false;
    car1/alarms/AlarmD1L/resetKey AT 461 : BOOL := false;
    car1/alarms/AlarmD1L/alarm AT 64 : BOOL := false;
    car1/alarms/AlarmD1L/i_rs1 AT 583 : DINT := 0;
    car1/alarms/AlarmD2L/enableAlarm AT 460 : BOOL := false;
    car1/alarms/AlarmD2L/resetKey AT 459 : BOOL := false;
    car1/alarms/AlarmD2L/alarm AT 63 : BOOL := false;
    car1/alarms/AlarmD2L/i_rs1 AT 585 : DINT := 0;
    car1/alarms/AlarmD3L/enableAlarm AT 458 : BOOL := false;
    car1/alarms/AlarmD3L/resetKey AT 457 : BOOL := false;
    car1/alarms/AlarmD3L/alarm AT 62 : BOOL := false;
    car1/alarms/AlarmD3L/i_rs1 AT 587 : DINT := 0;
    car1/alarms/AlarmD1R/enableAlarm AT 456 : BOOL := false;
    car1/alarms/AlarmD1R/resetKey AT 455 : BOOL := false;
    car1/alarms/AlarmD1R/alarm AT 61 : BOOL := false;
    car1/alarms/AlarmD1R/i_rs1 AT 589 : DINT := 0;
    car1/alarms/AlarmD2R/enableAlarm AT 454 : BOOL := false;
    car1/alarms/AlarmD2R/resetKey AT 453 : BOOL := false;
    car1/alarms/AlarmD2R/alarm AT 60 : BOOL := false;
    car1/alarms/AlarmD2R/i_rs1 AT 591 : DINT := 0;
    car1/alarms/AlarmD3R/enableAlarm AT 452 : BOOL := false;
    car1/alarms/AlarmD3R/resetKey AT 451 : BOOL := false;
    car1/alarms/AlarmD3R/alarm AT 59 : BOOL := false;
    car1/alarms/AlarmD3R/i_rs1 AT 593 : DINT := 0;
    car1/doorL1/compressedAir AT 56 : REAL := 200.0;
    car1/doorL1/cmdSupply AT 446 : BOOL := true;
    car1/doorL1/sensorSupply AT 445 : BOOL := true;
    car1/doorL1/enableOpening AT 447 : BOOL := false;
    car1/doorL1/enableClosing AT 448 : BOOL := false;
    car1/doorL1/closedDoorState AT 76 : BOOL := false;
    car1/doorL1/openedDoorState AT 75 : BOOL := false;
    car1/doorL1/faultState AT 546 : DINT := 0;
    car1/doorL1/doorPB/doorPB AT 475 : BOOL := false;
    car1/doorL1/doorPB/button AT 479 : BOOL := false;
    car1/doorL1/doorPB/_X_10 AT 480 : BOOL := true;
    car1/doorL1/doorPB/_X_11 AT 481 : BOOL := false;
    car1/doorL1/doorPB/_X_12 AT 482 : BOOL := false;
    car1/doorL1/doorLocking/lockingCmd AT 469 : BOOL := false;
    car1/doorL1/doorLocking/unlockingCmd AT 470 : BOOL := false;
    car1/doorL1/doorLocking/doorLocked AT 473 : BOOL := false;
    car1/doorL1/doorLocking/doorUnlocked AT 474 : BOOL := false;
    car1/doorL1/doorLocking/lockActive AT 478 : BOOL := false;
    car1/doorL1/doorLocking/i_rs1 AT 596 : DINT := 0;
    car1/doorL1/doorLocking/d_unlockedSensor AT 484 : BOOL := false;
    car1/doorL1/doorLocking/v_d_unlockedSensor AT 485 : BOOL := false;
    car1/doorL1/doorLocking/d_lockedSensor AT 486 : BOOL := false;
    car1/doorL1/doorLocking/v_d_lockedSensor AT 487 : BOOL := false;
    car1/doorL1/doorControlPart/enableOpening AT 447 : BOOL := false;
    car1/doorL1/doorControlPart/enableClosing AT 448 : BOOL := false;
    car1/doorL1/doorControlPart/openedDoor AT 471 : BOOL := false;
    car1/doorL1/doorControlPart/closedDoor AT 472 : BOOL := false;
    car1/doorL1/doorControlPart/lockedDoor AT 473 : BOOL := false;
    car1/doorL1/doorControlPart/unlockedDoor AT 474 : BOOL := false;
    car1/doorL1/doorControlPart/openingRequest AT 475 : BOOL := false;
    car1/doorL1/doorControlPart/doorOpeningCmd AT 476 : BOOL := false;
    car1/doorL1/doorControlPart/doorClosingCmd AT 477 : BOOL := false;
    car1/doorL1/doorControlPart/doorLockingCmd AT 469 : BOOL := false;
    car1/doorL1/doorControlPart/doorUnlockingCmd AT 470 : BOOL := false;
    car1/doorL1/doorControlPart/closedDoorState AT 76 : BOOL := false;
    car1/doorL1/doorControlPart/openedDoorState AT 75 : BOOL := false;
    car1/doorL1/doorControlPart/faultState AT 546 : DINT := 0;
    car1/doorL1/doorControlPart/_X_10 AT 489 : BOOL := true;
    car1/doorL1/doorControlPart/_X_11 AT 490 : BOOL := false;
    car1/doorL1/doorControlPart/_X_12 AT 491 : BOOL := false;
    car1/doorL1/doorControlPart/_X_13 AT 492 : BOOL := false;
    car1/doorL1/doorControlPart/_X_14 AT 493 : BOOL := false;
    car1/doorL1/doorControlPart/_X_15 AT 494 : BOOL := false;
    car1/doorL1/doorControlPart/_X_16 AT 495 : BOOL := false;
    car1/doorL1/door/compressedAir AT 56 : REAL := 200.0;
    car1/doorL1/door/cmdSupply AT 446 : BOOL := true;
    car1/doorL1/door/sensorSupply AT 445 : BOOL := true;
    car1/doorL1/door/openDoorCmd AT 476 : BOOL := false;
    car1/doorL1/door/closeDoorCmd AT 477 : BOOL := false;
    car1/doorL1/door/lockActive AT 478 : BOOL := false;
    car1/doorL1/door/doorOpened AT 471 : BOOL := false;
    car1/doorL1/door/doorClosed AT 472 : BOOL := false;
    car1/doorL1/door/increment AT 57 : REAL := 0.0;
    car1/doorL1/door/openDoor AT 502 : BOOL := false;
    car1/doorL1/door/closeDoor AT 503 : BOOL := false;
    car1/doorL1/door/doorPosition AT 58 : REAL := 0.0;
    car1/doorL1/door/length AT 59 : REAL := 1000.0;
    car1/doorL1/door/doorClosedSensorLogic AT 504 : BOOL := true;
    car1/doorL1/door/doorOpenedSensorLogic AT 505 : BOOL := true;
    car1/doorL1/door/d_locking AT 506 : BOOL := false;
    car1/doorL1/door/v_d_locking AT 60 : REAL := 50.0;
    car1/doorL1/door/d_doorClosedSensor AT 507 : BOOL := false;
    car1/doorL1/door/v_d_doorClosedSensor AT 508 : BOOL := false;
    car1/doorL1/door/d_doorOpenedSensor AT 509 : BOOL := false;
    car1/doorL1/door/v_d_doorOpenedSensor AT 510 : BOOL := false;
    car1/doorL2/compressedAir AT 55 : REAL := 200.0;
    car1/doorL2/cmdSupply AT 444 : BOOL := true;
    car1/doorL2/sensorSupply AT 443 : BOOL := true;
    car1/doorL2/enableOpening AT 447 : BOOL := false;
    car1/doorL2/enableClosing AT 448 : BOOL := false;
    car1/doorL2/closedDoorState AT 74 : BOOL := false;
    car1/doorL2/openedDoorState AT 73 : BOOL := false;
    car1/doorL2/faultState AT 545 : DINT := 0;
    car1/doorL2/doorPB/doorPB AT 517 : BOOL := false;
    car1/doorL2/doorPB/button AT 521 : BOOL := false;
    car1/doorL2/doorPB/_X_10 AT 522 : BOOL := true;
    car1/doorL2/doorPB/_X_11 AT 523 : BOOL := false;
    car1/doorL2/doorPB/_X_12 AT 524 : BOOL := false;
    car1/doorL2/doorLocking/lockingCmd AT 511 : BOOL := false;
    car1/doorL2/doorLocking/unlockingCmd AT 512 : BOOL := false;
    car1/doorL2/doorLocking/doorLocked AT 515 : BOOL := false;
    car1/doorL2/doorLocking/doorUnlocked AT 516 : BOOL := false;
    car1/doorL2/doorLocking/lockActive AT 520 : BOOL := false;
    car1/doorL2/doorLocking/i_rs1 AT 599 : DINT := 0;
    car1/doorL2/doorLocking/d_unlockedSensor AT 526 : BOOL := false;
    car1/doorL2/doorLocking/v_d_unlockedSensor AT 527 : BOOL := false;
    car1/doorL2/doorLocking/d_lockedSensor AT 528 : BOOL := false;
    car1/doorL2/doorLocking/v_d_lockedSensor AT 529 : BOOL := false;
    car1/doorL2/doorControlPart/enableOpening AT 447 : BOOL := false;
    car1/doorL2/doorControlPart/enableClosing AT 448 : BOOL := false;
    car1/doorL2/doorControlPart/openedDoor AT 513 : BOOL := false;
    car1/doorL2/doorControlPart/closedDoor AT 514 : BOOL := false;
    car1/doorL2/doorControlPart/lockedDoor AT 515 : BOOL := false;
    car1/doorL2/doorControlPart/unlockedDoor AT 516 : BOOL := false;
    car1/doorL2/doorControlPart/openingRequest AT 517 : BOOL := false;
    car1/doorL2/doorControlPart/doorOpeningCmd AT 518 : BOOL := false;
    car1/doorL2/doorControlPart/doorClosingCmd AT 519 : BOOL := false;
    car1/doorL2/doorControlPart/doorLockingCmd AT 511 : BOOL := false;
    car1/doorL2/doorControlPart/doorUnlockingCmd AT 512 : BOOL := false;
    car1/doorL2/doorControlPart/closedDoorState AT 74 : BOOL := false;
    car1/doorL2/doorControlPart/openedDoorState AT 73 : BOOL := false;
    car1/doorL2/doorControlPart/faultState AT 545 : DINT := 0;
    car1/doorL2/doorControlPart/_X_10 AT 531 : BOOL := true;
    car1/doorL2/doorControlPart/_X_11 AT 532 : BOOL := false;
    car1/doorL2/doorControlPart/_X_12 AT 533 : BOOL := false;
    car1/doorL2/doorControlPart/_X_13 AT 534 : BOOL := false;
    car1/doorL2/doorControlPart/_X_14 AT 535 : BOOL := false;
    car1/doorL2/doorControlPart/_X_15 AT 536 : BOOL := false;
    car1/doorL2/doorControlPart/_X_16 AT 537 : BOOL := false;
    car1/doorL2/door/compressedAir AT 55 : REAL := 200.0;
    car1/doorL2/door/cmdSupply AT 444 : BOOL := true;
    car1/doorL2/door/sensorSupply AT 443 : BOOL := true;
    car1/doorL2/door/openDoorCmd AT 518 : BOOL := false;
    car1/doorL2/door/closeDoorCmd AT 519 : BOOL := false;
    car1/doorL2/door/lockActive AT 520 : BOOL := false;
    car1/doorL2/door/doorOpened AT 513 : BOOL := false;
    car1/doorL2/door/doorClosed AT 514 : BOOL := false;
    car1/doorL2/door/increment AT 61 : REAL := 0.0;
    car1/doorL2/door/openDoor AT 544 : BOOL := false;
    car1/doorL2/door/closeDoor AT 545 : BOOL := false;
    car1/doorL2/door/doorPosition AT 62 : REAL := 0.0;
    car1/doorL2/door/length AT 63 : REAL := 1000.0;
    car1/doorL2/door/doorClosedSensorLogic AT 546 : BOOL := true;
    car1/doorL2/door/doorOpenedSensorLogic AT 547 : BOOL := true;
    car1/doorL2/door/d_locking AT 548 : BOOL := false;
    car1/doorL2/door/v_d_locking AT 64 : REAL := 50.0;
    car1/doorL2/door/d_doorClosedSensor AT 549 : BOOL := false;
    car1/doorL2/door/v_d_doorClosedSensor AT 550 : BOOL := false;
    car1/doorL2/door/d_doorOpenedSensor AT 551 : BOOL := false;
    car1/doorL2/door/v_d_doorOpenedSensor AT 552 : BOOL := false;
    car1/doorL3/compressedAir AT 54 : REAL := 200.0;
    car1/doorL3/cmdSupply AT 442 : BOOL := true;
    car1/doorL3/sensorSupply AT 441 : BOOL := true;
    car1/doorL3/enableOpening AT 447 : BOOL := false;
    car1/doorL3/enableClosing AT 448 : BOOL := false;
    car1/doorL3/closedDoorState AT 72 : BOOL := false;
    car1/doorL3/openedDoorState AT 71 : BOOL := false;
    car1/doorL3/faultState AT 544 : DINT := 0;
    car1/doorL3/doorPB/doorPB AT 559 : BOOL := false;
    car1/doorL3/doorPB/button AT 563 : BOOL := false;
    car1/doorL3/doorPB/_X_10 AT 564 : BOOL := true;
    car1/doorL3/doorPB/_X_11 AT 565 : BOOL := false;
    car1/doorL3/doorPB/_X_12 AT 566 : BOOL := false;
    car1/doorL3/doorLocking/lockingCmd AT 553 : BOOL := false;
    car1/doorL3/doorLocking/unlockingCmd AT 554 : BOOL := false;
    car1/doorL3/doorLocking/doorLocked AT 557 : BOOL := false;
    car1/doorL3/doorLocking/doorUnlocked AT 558 : BOOL := false;
    car1/doorL3/doorLocking/lockActive AT 562 : BOOL := false;
    car1/doorL3/doorLocking/i_rs1 AT 602 : DINT := 0;
    car1/doorL3/doorLocking/d_unlockedSensor AT 568 : BOOL := false;
    car1/doorL3/doorLocking/v_d_unlockedSensor AT 569 : BOOL := false;
    car1/doorL3/doorLocking/d_lockedSensor AT 570 : BOOL := false;
    car1/doorL3/doorLocking/v_d_lockedSensor AT 571 : BOOL := false;
    car1/doorL3/doorControlPart/enableOpening AT 447 : BOOL := false;
    car1/doorL3/doorControlPart/enableClosing AT 448 : BOOL := false;
    car1/doorL3/doorControlPart/openedDoor AT 555 : BOOL := false;
    car1/doorL3/doorControlPart/closedDoor AT 556 : BOOL := false;
    car1/doorL3/doorControlPart/lockedDoor AT 557 : BOOL := false;
    car1/doorL3/doorControlPart/unlockedDoor AT 558 : BOOL := false;
    car1/doorL3/doorControlPart/openingRequest AT 559 : BOOL := false;
    car1/doorL3/doorControlPart/doorOpeningCmd AT 560 : BOOL := false;
    car1/doorL3/doorControlPart/doorClosingCmd AT 561 : BOOL := false;
    car1/doorL3/doorControlPart/doorLockingCmd AT 553 : BOOL := false;
    car1/doorL3/doorControlPart/doorUnlockingCmd AT 554 : BOOL := false;
    car1/doorL3/doorControlPart/closedDoorState AT 72 : BOOL := false;
    car1/doorL3/doorControlPart/openedDoorState AT 71 : BOOL := false;
    car1/doorL3/doorControlPart/faultState AT 544 : DINT := 0;
    car1/doorL3/doorControlPart/_X_10 AT 573 : BOOL := true;
    car1/doorL3/doorControlPart/_X_11 AT 574 : BOOL := false;
    car1/doorL3/doorControlPart/_X_12 AT 575 : BOOL := false;
    car1/doorL3/doorControlPart/_X_13 AT 576 : BOOL := false;
    car1/doorL3/doorControlPart/_X_14 AT 577 : BOOL := false;
    car1/doorL3/doorControlPart/_X_15 AT 578 : BOOL := false;
    car1/doorL3/doorControlPart/_X_16 AT 579 : BOOL := false;
    car1/doorL3/door/compressedAir AT 54 : REAL := 200.0;
    car1/doorL3/door/cmdSupply AT 442 : BOOL := true;
    car1/doorL3/door/sensorSupply AT 441 : BOOL := true;
    car1/doorL3/door/openDoorCmd AT 560 : BOOL := false;
    car1/doorL3/door/closeDoorCmd AT 561 : BOOL := false;
    car1/doorL3/door/lockActive AT 562 : BOOL := false;
    car1/doorL3/door/doorOpened AT 555 : BOOL := false;
    car1/doorL3/door/doorClosed AT 556 : BOOL := false;
    car1/doorL3/door/increment AT 65 : REAL := 0.0;
    car1/doorL3/door/openDoor AT 586 : BOOL := false;
    car1/doorL3/door/closeDoor AT 587 : BOOL := false;
    car1/doorL3/door/doorPosition AT 66 : REAL := 0.0;
    car1/doorL3/door/length AT 67 : REAL := 1000.0;
    car1/doorL3/door/doorClosedSensorLogic AT 588 : BOOL := true;
    car1/doorL3/door/doorOpenedSensorLogic AT 589 : BOOL := true;
    car1/doorL3/door/d_locking AT 590 : BOOL := false;
    car1/doorL3/door/v_d_locking AT 68 : REAL := 50.0;
    car1/doorL3/door/d_doorClosedSensor AT 591 : BOOL := false;
    car1/doorL3/door/v_d_doorClosedSensor AT 592 : BOOL := false;
    car1/doorL3/door/d_doorOpenedSensor AT 593 : BOOL := false;
    car1/doorL3/door/v_d_doorOpenedSensor AT 594 : BOOL := false;
    car1/doorR1/compressedAir AT 53 : REAL := 200.0;
    car1/doorR1/cmdSupply AT 440 : BOOL := true;
    car1/doorR1/sensorSupply AT 439 : BOOL := true;
    car1/doorR1/enableOpening AT 449 : BOOL := false;
    car1/doorR1/enableClosing AT 450 : BOOL := false;
    car1/doorR1/closedDoorState AT 70 : BOOL := false;
    car1/doorR1/openedDoorState AT 69 : BOOL := false;
    car1/doorR1/faultState AT 543 : DINT := 0;
    car1/doorR1/doorPB/doorPB AT 601 : BOOL := false;
    car1/doorR1/doorPB/button AT 605 : BOOL := false;
    car1/doorR1/doorPB/_X_10 AT 606 : BOOL := true;
    car1/doorR1/doorPB/_X_11 AT 607 : BOOL := false;
    car1/doorR1/doorPB/_X_12 AT 608 : BOOL := false;
    car1/doorR1/doorLocking/lockingCmd AT 595 : BOOL := false;
    car1/doorR1/doorLocking/unlockingCmd AT 596 : BOOL := false;
    car1/doorR1/doorLocking/doorLocked AT 599 : BOOL := false;
    car1/doorR1/doorLocking/doorUnlocked AT 600 : BOOL := false;
    car1/doorR1/doorLocking/lockActive AT 604 : BOOL := false;
    car1/doorR1/doorLocking/i_rs1 AT 605 : DINT := 0;
    car1/doorR1/doorLocking/d_unlockedSensor AT 610 : BOOL := false;
    car1/doorR1/doorLocking/v_d_unlockedSensor AT 611 : BOOL := false;
    car1/doorR1/doorLocking/d_lockedSensor AT 612 : BOOL := false;
    car1/doorR1/doorLocking/v_d_lockedSensor AT 613 : BOOL := false;
    car1/doorR1/doorControlPart/enableOpening AT 449 : BOOL := false;
    car1/doorR1/doorControlPart/enableClosing AT 450 : BOOL := false;
    car1/doorR1/doorControlPart/openedDoor AT 597 : BOOL := false;
    car1/doorR1/doorControlPart/closedDoor AT 598 : BOOL := false;
    car1/doorR1/doorControlPart/lockedDoor AT 599 : BOOL := false;
    car1/doorR1/doorControlPart/unlockedDoor AT 600 : BOOL := false;
    car1/doorR1/doorControlPart/openingRequest AT 601 : BOOL := false;
    car1/doorR1/doorControlPart/doorOpeningCmd AT 602 : BOOL := false;
    car1/doorR1/doorControlPart/doorClosingCmd AT 603 : BOOL := false;
    car1/doorR1/doorControlPart/doorLockingCmd AT 595 : BOOL := false;
    car1/doorR1/doorControlPart/doorUnlockingCmd AT 596 : BOOL := false;
    car1/doorR1/doorControlPart/closedDoorState AT 70 : BOOL := false;
    car1/doorR1/doorControlPart/openedDoorState AT 69 : BOOL := false;
    car1/doorR1/doorControlPart/faultState AT 543 : DINT := 0;
    car1/doorR1/doorControlPart/_X_10 AT 615 : BOOL := true;
    car1/doorR1/doorControlPart/_X_11 AT 616 : BOOL := false;
    car1/doorR1/doorControlPart/_X_12 AT 617 : BOOL := false;
    car1/doorR1/doorControlPart/_X_13 AT 618 : BOOL := false;
    car1/doorR1/doorControlPart/_X_14 AT 619 : BOOL := false;
    car1/doorR1/doorControlPart/_X_15 AT 620 : BOOL := false;
    car1/doorR1/doorControlPart/_X_16 AT 621 : BOOL := false;
    car1/doorR1/door/compressedAir AT 53 : REAL := 200.0;
    car1/doorR1/door/cmdSupply AT 440 : BOOL := true;
    car1/doorR1/door/sensorSupply AT 439 : BOOL := true;
    car1/doorR1/door/openDoorCmd AT 602 : BOOL := false;
    car1/doorR1/door/closeDoorCmd AT 603 : BOOL := false;
    car1/doorR1/door/lockActive AT 604 : BOOL := false;
    car1/doorR1/door/doorOpened AT 597 : BOOL := false;
    car1/doorR1/door/doorClosed AT 598 : BOOL := false;
    car1/doorR1/door/increment AT 69 : REAL := 0.0;
    car1/doorR1/door/openDoor AT 628 : BOOL := false;
    car1/doorR1/door/closeDoor AT 629 : BOOL := false;
    car1/doorR1/door/doorPosition AT 70 : REAL := 0.0;
    car1/doorR1/door/length AT 71 : REAL := 1000.0;
    car1/doorR1/door/doorClosedSensorLogic AT 630 : BOOL := true;
    car1/doorR1/door/doorOpenedSensorLogic AT 631 : BOOL := true;
    car1/doorR1/door/d_locking AT 632 : BOOL := false;
    car1/doorR1/door/v_d_locking AT 72 : REAL := 50.0;
    car1/doorR1/door/d_doorClosedSensor AT 633 : BOOL := false;
    car1/doorR1/door/v_d_doorClosedSensor AT 634 : BOOL := false;
    car1/doorR1/door/d_doorOpenedSensor AT 635 : BOOL := false;
    car1/doorR1/door/v_d_doorOpenedSensor AT 636 : BOOL := false;
    car1/doorR2/compressedAir AT 52 : REAL := 200.0;
    car1/doorR2/cmdSupply AT 438 : BOOL := true;
    car1/doorR2/sensorSupply AT 437 : BOOL := true;
    car1/doorR2/enableOpening AT 449 : BOOL := false;
    car1/doorR2/enableClosing AT 450 : BOOL := false;
    car1/doorR2/closedDoorState AT 68 : BOOL := false;
    car1/doorR2/openedDoorState AT 67 : BOOL := false;
    car1/doorR2/faultState AT 542 : DINT := 0;
    car1/doorR2/doorPB/doorPB AT 643 : BOOL := false;
    car1/doorR2/doorPB/button AT 647 : BOOL := false;
    car1/doorR2/doorPB/_X_10 AT 648 : BOOL := true;
    car1/doorR2/doorPB/_X_11 AT 649 : BOOL := false;
    car1/doorR2/doorPB/_X_12 AT 650 : BOOL := false;
    car1/doorR2/doorLocking/lockingCmd AT 637 : BOOL := false;
    car1/doorR2/doorLocking/unlockingCmd AT 638 : BOOL := false;
    car1/doorR2/doorLocking/doorLocked AT 641 : BOOL := false;
    car1/doorR2/doorLocking/doorUnlocked AT 642 : BOOL := false;
    car1/doorR2/doorLocking/lockActive AT 646 : BOOL := false;
    car1/doorR2/doorLocking/i_rs1 AT 608 : DINT := 0;
    car1/doorR2/doorLocking/d_unlockedSensor AT 652 : BOOL := false;
    car1/doorR2/doorLocking/v_d_unlockedSensor AT 653 : BOOL := false;
    car1/doorR2/doorLocking/d_lockedSensor AT 654 : BOOL := false;
    car1/doorR2/doorLocking/v_d_lockedSensor AT 655 : BOOL := false;
    car1/doorR2/doorControlPart/enableOpening AT 449 : BOOL := false;
    car1/doorR2/doorControlPart/enableClosing AT 450 : BOOL := false;
    car1/doorR2/doorControlPart/openedDoor AT 639 : BOOL := false;
    car1/doorR2/doorControlPart/closedDoor AT 640 : BOOL := false;
    car1/doorR2/doorControlPart/lockedDoor AT 641 : BOOL := false;
    car1/doorR2/doorControlPart/unlockedDoor AT 642 : BOOL := false;
    car1/doorR2/doorControlPart/openingRequest AT 643 : BOOL := false;
    car1/doorR2/doorControlPart/doorOpeningCmd AT 644 : BOOL := false;
    car1/doorR2/doorControlPart/doorClosingCmd AT 645 : BOOL := false;
    car1/doorR2/doorControlPart/doorLockingCmd AT 637 : BOOL := false;
    car1/doorR2/doorControlPart/doorUnlockingCmd AT 638 : BOOL := false;
    car1/doorR2/doorControlPart/closedDoorState AT 68 : BOOL := false;
    car1/doorR2/doorControlPart/openedDoorState AT 67 : BOOL := false;
    car1/doorR2/doorControlPart/faultState AT 542 : DINT := 0;
    car1/doorR2/doorControlPart/_X_10 AT 657 : BOOL := true;
    car1/doorR2/doorControlPart/_X_11 AT 658 : BOOL := false;
    car1/doorR2/doorControlPart/_X_12 AT 659 : BOOL := false;
    car1/doorR2/doorControlPart/_X_13 AT 660 : BOOL := false;
    car1/doorR2/doorControlPart/_X_14 AT 661 : BOOL := false;
    car1/doorR2/doorControlPart/_X_15 AT 662 : BOOL := false;
    car1/doorR2/doorControlPart/_X_16 AT 663 : BOOL := false;
    car1/doorR2/door/compressedAir AT 52 : REAL := 200.0;
    car1/doorR2/door/cmdSupply AT 438 : BOOL := true;
    car1/doorR2/door/sensorSupply AT 437 : BOOL := true;
    car1/doorR2/door/openDoorCmd AT 644 : BOOL := false;
    car1/doorR2/door/closeDoorCmd AT 645 : BOOL := false;
    car1/doorR2/door/lockActive AT 646 : BOOL := false;
    car1/doorR2/door/doorOpened AT 639 : BOOL := false;
    car1/doorR2/door/doorClosed AT 640 : BOOL := false;
    car1/doorR2/door/increment AT 73 : REAL := 0.0;
    car1/doorR2/door/openDoor AT 670 : BOOL := false;
    car1/doorR2/door/closeDoor AT 671 : BOOL := false;
    car1/doorR2/door/doorPosition AT 74 : REAL := 0.0;
    car1/doorR2/door/length AT 75 : REAL := 1000.0;
    car1/doorR2/door/doorClosedSensorLogic AT 672 : BOOL := true;
    car1/doorR2/door/doorOpenedSensorLogic AT 673 : BOOL := true;
    car1/doorR2/door/d_locking AT 674 : BOOL := false;
    car1/doorR2/door/v_d_locking AT 76 : REAL := 50.0;
    car1/doorR2/door/d_doorClosedSensor AT 675 : BOOL := false;
    car1/doorR2/door/v_d_doorClosedSensor AT 676 : BOOL := false;
    car1/doorR2/door/d_doorOpenedSensor AT 677 : BOOL := false;
    car1/doorR2/door/v_d_doorOpenedSensor AT 678 : BOOL := false;
    car1/doorR3/compressedAir AT 51 : REAL := 200.0;
    car1/doorR3/cmdSupply AT 436 : BOOL := true;
    car1/doorR3/sensorSupply AT 435 : BOOL := true;
    car1/doorR3/enableOpening AT 449 : BOOL := false;
    car1/doorR3/enableClosing AT 450 : BOOL := false;
    car1/doorR3/closedDoorState AT 66 : BOOL := false;
    car1/doorR3/openedDoorState AT 65 : BOOL := false;
    car1/doorR3/faultState AT 541 : DINT := 0;
    car1/doorR3/doorPB/doorPB AT 685 : BOOL := false;
    car1/doorR3/doorPB/button AT 689 : BOOL := false;
    car1/doorR3/doorPB/_X_10 AT 690 : BOOL := true;
    car1/doorR3/doorPB/_X_11 AT 691 : BOOL := false;
    car1/doorR3/doorPB/_X_12 AT 692 : BOOL := false;
    car1/doorR3/doorLocking/lockingCmd AT 679 : BOOL := false;
    car1/doorR3/doorLocking/unlockingCmd AT 680 : BOOL := false;
    car1/doorR3/doorLocking/doorLocked AT 683 : BOOL := false;
    car1/doorR3/doorLocking/doorUnlocked AT 684 : BOOL := false;
    car1/doorR3/doorLocking/lockActive AT 688 : BOOL := false;
    car1/doorR3/doorLocking/i_rs1 AT 611 : DINT := 0;
    car1/doorR3/doorLocking/d_unlockedSensor AT 694 : BOOL := false;
    car1/doorR3/doorLocking/v_d_unlockedSensor AT 695 : BOOL := false;
    car1/doorR3/doorLocking/d_lockedSensor AT 696 : BOOL := false;
    car1/doorR3/doorLocking/v_d_lockedSensor AT 697 : BOOL := false;
    car1/doorR3/doorControlPart/enableOpening AT 449 : BOOL := false;
    car1/doorR3/doorControlPart/enableClosing AT 450 : BOOL := false;
    car1/doorR3/doorControlPart/openedDoor AT 681 : BOOL := false;
    car1/doorR3/doorControlPart/closedDoor AT 682 : BOOL := false;
    car1/doorR3/doorControlPart/lockedDoor AT 683 : BOOL := false;
    car1/doorR3/doorControlPart/unlockedDoor AT 684 : BOOL := false;
    car1/doorR3/doorControlPart/openingRequest AT 685 : BOOL := false;
    car1/doorR3/doorControlPart/doorOpeningCmd AT 686 : BOOL := false;
    car1/doorR3/doorControlPart/doorClosingCmd AT 687 : BOOL := false;
    car1/doorR3/doorControlPart/doorLockingCmd AT 679 : BOOL := false;
    car1/doorR3/doorControlPart/doorUnlockingCmd AT 680 : BOOL := false;
    car1/doorR3/doorControlPart/closedDoorState AT 66 : BOOL := false;
    car1/doorR3/doorControlPart/openedDoorState AT 65 : BOOL := false;
    car1/doorR3/doorControlPart/faultState AT 541 : DINT := 0;
    car1/doorR3/doorControlPart/_X_10 AT 699 : BOOL := true;
    car1/doorR3/doorControlPart/_X_11 AT 700 : BOOL := false;
    car1/doorR3/doorControlPart/_X_12 AT 701 : BOOL := false;
    car1/doorR3/doorControlPart/_X_13 AT 702 : BOOL := false;
    car1/doorR3/doorControlPart/_X_14 AT 703 : BOOL := false;
    car1/doorR3/doorControlPart/_X_15 AT 704 : BOOL := false;
    car1/doorR3/doorControlPart/_X_16 AT 705 : BOOL := false;
    car1/doorR3/door/compressedAir AT 51 : REAL := 200.0;
    car1/doorR3/door/cmdSupply AT 436 : BOOL := true;
    car1/doorR3/door/sensorSupply AT 435 : BOOL := true;
    car1/doorR3/door/openDoorCmd AT 686 : BOOL := false;
    car1/doorR3/door/closeDoorCmd AT 687 : BOOL := false;
    car1/doorR3/door/lockActive AT 688 : BOOL := false;
    car1/doorR3/door/doorOpened AT 681 : BOOL := false;
    car1/doorR3/door/doorClosed AT 682 : BOOL := false;
    car1/doorR3/door/increment AT 77 : REAL := 0.0;
    car1/doorR3/door/openDoor AT 712 : BOOL := false;
    car1/doorR3/door/closeDoor AT 713 : BOOL := false;
    car1/doorR3/door/doorPosition AT 78 : REAL := 0.0;
    car1/doorR3/door/length AT 79 : REAL := 1000.0;
    car1/doorR3/door/doorClosedSensorLogic AT 714 : BOOL := true;
    car1/doorR3/door/doorOpenedSensorLogic AT 715 : BOOL := true;
    car1/doorR3/door/d_locking AT 716 : BOOL := false;
    car1/doorR3/door/v_d_locking AT 80 : REAL := 50.0;
    car1/doorR3/door/d_doorClosedSensor AT 717 : BOOL := false;
    car1/doorR3/door/v_d_doorClosedSensor AT 718 : BOOL := false;
    car1/doorR3/door/d_doorOpenedSensor AT 719 : BOOL := false;
    car1/doorR3/door/v_d_doorOpenedSensor AT 720 : BOOL := false;
    car2/AuthorizationClosingLeftC1 AT 101 : BOOL := false;
    car2/AuthorizationOpeningRightC1 AT 102 : BOOL := false;
    car2/AuthorizationClosingRightC1 AT 103 : BOOL := false;
    car2/AuthorizationOpeningLeftC1 AT 104 : BOOL := false;
    car2/AuthorizationClosingLeftC2 AT 105 : BOOL := false;
    car2/AuthorizationOpeningRightC2 AT 106 : BOOL := false;
    car2/AuthorizationClosingRightC2 AT 107 : BOOL := false;
    car2/AuthorizationOpeningLeftC2 AT 108 : BOOL := false;
    car2/doorL1Closed AT 58 : BOOL := false;
    car2/doorL1Opened AT 57 : BOOL := false;
    car2/doorL1Fault AT 540 : DINT := 0;
    car2/doorL2Closed AT 56 : BOOL := false;
    car2/doorL2Opened AT 55 : BOOL := false;
    car2/doorL2Fault AT 539 : DINT := 0;
    car2/doorL3Closed AT 54 : BOOL := false;
    car2/doorL3Opened AT 53 : BOOL := false;
    car2/doorL3Fault AT 538 : DINT := 0;
    car2/doorR1Closed AT 52 : BOOL := false;
    car2/doorR1Opened AT 51 : BOOL := false;
    car2/doorR1Fault AT 537 : DINT := 0;
    car2/doorR2Closed AT 50 : BOOL := false;
    car2/doorR2Opened AT 49 : BOOL := false;
    car2/doorR2Fault AT 536 : DINT := 0;
    car2/doorR3Closed AT 48 : BOOL := false;
    car2/doorR3Opened AT 47 : BOOL := false;
    car2/doorR3Fault AT 535 : DINT := 0;
    car2/AlarmD1L AT 46 : BOOL := false;
    car2/AlarmD2L AT 45 : BOOL := false;
    car2/AlarmD3L AT 44 : BOOL := false;
    car2/AlarmD1R AT 43 : BOOL := false;
    car2/AlarmD2R AT 42 : BOOL := false;
    car2/AlarmD3R AT 41 : BOOL := false;
    car2/authorizations/AuthorizationClosingLeftC1 AT 101 : BOOL := false;
    car2/authorizations/AuthorizationOpeningRightC1 AT 102 : BOOL := false;
    car2/authorizations/AuthorizationClosingRightC1 AT 103 : BOOL := false;
    car2/authorizations/AuthorizationOpeningLeftC1 AT 104 : BOOL := false;
    car2/authorizations/AuthorizationClosingLeftC2 AT 105 : BOOL := false;
    car2/authorizations/AuthorizationOpeningRightC2 AT 106 : BOOL := false;
    car2/authorizations/AuthorizationClosingRightC2 AT 107 : BOOL := false;
    car2/authorizations/AuthorizationOpeningLeftC2 AT 108 : BOOL := false;
    car2/authorizations/AuthorizationOpeningLeft AT 733 : BOOL := false;
    car2/authorizations/AuthorizationClosingLeft AT 734 : BOOL := false;
    car2/authorizations/AuthorizationOpeningRight AT 735 : BOOL := false;
    car2/authorizations/AuthorizationClosingRight AT 736 : BOOL := false;
    car2/alarms/AlarmD1L AT 46 : BOOL := false;
    car2/alarms/AlarmD2L AT 45 : BOOL := false;
    car2/alarms/AlarmD3L AT 44 : BOOL := false;
    car2/alarms/AlarmD1R AT 43 : BOOL := false;
    car2/alarms/AlarmD2R AT 42 : BOOL := false;
    car2/alarms/AlarmD3R AT 41 : BOOL := false;
    car2/alarms/AlarmD1L/enableAlarm AT 748 : BOOL := false;
    car2/alarms/AlarmD1L/resetKey AT 747 : BOOL := false;
    car2/alarms/AlarmD1L/alarm AT 46 : BOOL := false;
    car2/alarms/AlarmD1L/i_rs1 AT 613 : DINT := 0;
    car2/alarms/AlarmD2L/enableAlarm AT 746 : BOOL := false;
    car2/alarms/AlarmD2L/resetKey AT 745 : BOOL := false;
    car2/alarms/AlarmD2L/alarm AT 45 : BOOL := false;
    car2/alarms/AlarmD2L/i_rs1 AT 615 : DINT := 0;
    car2/alarms/AlarmD3L/enableAlarm AT 744 : BOOL := false;
    car2/alarms/AlarmD3L/resetKey AT 743 : BOOL := false;
    car2/alarms/AlarmD3L/alarm AT 44 : BOOL := false;
    car2/alarms/AlarmD3L/i_rs1 AT 617 : DINT := 0;
    car2/alarms/AlarmD1R/enableAlarm AT 742 : BOOL := false;
    car2/alarms/AlarmD1R/resetKey AT 741 : BOOL := false;
    car2/alarms/AlarmD1R/alarm AT 43 : BOOL := false;
    car2/alarms/AlarmD1R/i_rs1 AT 619 : DINT := 0;
    car2/alarms/AlarmD2R/enableAlarm AT 740 : BOOL := false;
    car2/alarms/AlarmD2R/resetKey AT 739 : BOOL := false;
    car2/alarms/AlarmD2R/alarm AT 42 : BOOL := false;
    car2/alarms/AlarmD2R/i_rs1 AT 621 : DINT := 0;
    car2/alarms/AlarmD3R/enableAlarm AT 738 : BOOL := false;
    car2/alarms/AlarmD3R/resetKey AT 737 : BOOL := false;
    car2/alarms/AlarmD3R/alarm AT 41 : BOOL := false;
    car2/alarms/AlarmD3R/i_rs1 AT 623 : DINT := 0;
    car2/doorL1/compressedAir AT 86 : REAL := 200.0;
    car2/doorL1/cmdSupply AT 732 : BOOL := true;
    car2/doorL1/sensorSupply AT 731 : BOOL := true;
    car2/doorL1/enableOpening AT 733 : BOOL := false;
    car2/doorL1/enableClosing AT 734 : BOOL := false;
    car2/doorL1/closedDoorState AT 58 : BOOL := false;
    car2/doorL1/openedDoorState AT 57 : BOOL := false;
    car2/doorL1/faultState AT 540 : DINT := 0;
    car2/doorL1/doorPB/doorPB AT 761 : BOOL := false;
    car2/doorL1/doorPB/button AT 765 : BOOL := false;
    car2/doorL1/doorPB/_X_10 AT 766 : BOOL := true;
    car2/doorL1/doorPB/_X_11 AT 767 : BOOL := false;
    car2/doorL1/doorPB/_X_12 AT 768 : BOOL := false;
    car2/doorL1/doorLocking/lockingCmd AT 755 : BOOL := false;
    car2/doorL1/doorLocking/unlockingCmd AT 756 : BOOL := false;
    car2/doorL1/doorLocking/doorLocked AT 759 : BOOL := false;
    car2/doorL1/doorLocking/doorUnlocked AT 760 : BOOL := false;
    car2/doorL1/doorLocking/lockActive AT 764 : BOOL := false;
    car2/doorL1/doorLocking/i_rs1 AT 626 : DINT := 0;
    car2/doorL1/doorLocking/d_unlockedSensor AT 770 : BOOL := false;
    car2/doorL1/doorLocking/v_d_unlockedSensor AT 771 : BOOL := false;
    car2/doorL1/doorLocking/d_lockedSensor AT 772 : BOOL := false;
    car2/doorL1/doorLocking/v_d_lockedSensor AT 773 : BOOL := false;
    car2/doorL1/doorControlPart/enableOpening AT 733 : BOOL := false;
    car2/doorL1/doorControlPart/enableClosing AT 734 : BOOL := false;
    car2/doorL1/doorControlPart/openedDoor AT 757 : BOOL := false;
    car2/doorL1/doorControlPart/closedDoor AT 758 : BOOL := false;
    car2/doorL1/doorControlPart/lockedDoor AT 759 : BOOL := false;
    car2/doorL1/doorControlPart/unlockedDoor AT 760 : BOOL := false;
    car2/doorL1/doorControlPart/openingRequest AT 761 : BOOL := false;
    car2/doorL1/doorControlPart/doorOpeningCmd AT 762 : BOOL := false;
    car2/doorL1/doorControlPart/doorClosingCmd AT 763 : BOOL := false;
    car2/doorL1/doorControlPart/doorLockingCmd AT 755 : BOOL := false;
    car2/doorL1/doorControlPart/doorUnlockingCmd AT 756 : BOOL := false;
    car2/doorL1/doorControlPart/closedDoorState AT 58 : BOOL := false;
    car2/doorL1/doorControlPart/openedDoorState AT 57 : BOOL := false;
    car2/doorL1/doorControlPart/faultState AT 540 : DINT := 0;
    car2/doorL1/doorControlPart/_X_10 AT 775 : BOOL := true;
    car2/doorL1/doorControlPart/_X_11 AT 776 : BOOL := false;
    car2/doorL1/doorControlPart/_X_12 AT 777 : BOOL := false;
    car2/doorL1/doorControlPart/_X_13 AT 778 : BOOL := false;
    car2/doorL1/doorControlPart/_X_14 AT 779 : BOOL := false;
    car2/doorL1/doorControlPart/_X_15 AT 780 : BOOL := false;
    car2/doorL1/doorControlPart/_X_16 AT 781 : BOOL := false;
    car2/doorL1/door/compressedAir AT 86 : REAL := 200.0;
    car2/doorL1/door/cmdSupply AT 732 : BOOL := true;
    car2/doorL1/door/sensorSupply AT 731 : BOOL := true;
    car2/doorL1/door/openDoorCmd AT 762 : BOOL := false;
    car2/doorL1/door/closeDoorCmd AT 763 : BOOL := false;
    car2/doorL1/door/lockActive AT 764 : BOOL := false;
    car2/doorL1/door/doorOpened AT 757 : BOOL := false;
    car2/doorL1/door/doorClosed AT 758 : BOOL := false;
    car2/doorL1/door/increment AT 87 : REAL := 0.0;
    car2/doorL1/door/openDoor AT 788 : BOOL := false;
    car2/doorL1/door/closeDoor AT 789 : BOOL := false;
    car2/doorL1/door/doorPosition AT 88 : REAL := 0.0;
    car2/doorL1/door/length AT 89 : REAL := 1000.0;
    car2/doorL1/door/doorClosedSensorLogic AT 790 : BOOL := true;
    car2/doorL1/door/doorOpenedSensorLogic AT 791 : BOOL := true;
    car2/doorL1/door/d_locking AT 792 : BOOL := false;
    car2/doorL1/door/v_d_locking AT 90 : REAL := 50.0;
    car2/doorL1/door/d_doorClosedSensor AT 793 : BOOL := false;
    car2/doorL1/door/v_d_doorClosedSensor AT 794 : BOOL := false;
    car2/doorL1/door/d_doorOpenedSensor AT 795 : BOOL := false;
    car2/doorL1/door/v_d_doorOpenedSensor AT 796 : BOOL := false;
    car2/doorL2/compressedAir AT 85 : REAL := 200.0;
    car2/doorL2/cmdSupply AT 730 : BOOL := true;
    car2/doorL2/sensorSupply AT 729 : BOOL := true;
    car2/doorL2/enableOpening AT 733 : BOOL := false;
    car2/doorL2/enableClosing AT 734 : BOOL := false;
    car2/doorL2/closedDoorState AT 56 : BOOL := false;
    car2/doorL2/openedDoorState AT 55 : BOOL := false;
    car2/doorL2/faultState AT 539 : DINT := 0;
    car2/doorL2/doorPB/doorPB AT 803 : BOOL := false;
    car2/doorL2/doorPB/button AT 807 : BOOL := false;
    car2/doorL2/doorPB/_X_10 AT 808 : BOOL := true;
    car2/doorL2/doorPB/_X_11 AT 809 : BOOL := false;
    car2/doorL2/doorPB/_X_12 AT 810 : BOOL := false;
    car2/doorL2/doorLocking/lockingCmd AT 797 : BOOL := false;
    car2/doorL2/doorLocking/unlockingCmd AT 798 : BOOL := false;
    car2/doorL2/doorLocking/doorLocked AT 801 : BOOL := false;
    car2/doorL2/doorLocking/doorUnlocked AT 802 : BOOL := false;
    car2/doorL2/doorLocking/lockActive AT 806 : BOOL := false;
    car2/doorL2/doorLocking/i_rs1 AT 629 : DINT := 0;
    car2/doorL2/doorLocking/d_unlockedSensor AT 812 : BOOL := false;
    car2/doorL2/doorLocking/v_d_unlockedSensor AT 813 : BOOL := false;
    car2/doorL2/doorLocking/d_lockedSensor AT 814 : BOOL := false;
    car2/doorL2/doorLocking/v_d_lockedSensor AT 815 : BOOL := false;
    car2/doorL2/doorControlPart/enableOpening AT 733 : BOOL := false;
    car2/doorL2/doorControlPart/enableClosing AT 734 : BOOL := false;
    car2/doorL2/doorControlPart/openedDoor AT 799 : BOOL := false;
    car2/doorL2/doorControlPart/closedDoor AT 800 : BOOL := false;
    car2/doorL2/doorControlPart/lockedDoor AT 801 : BOOL := false;
    car2/doorL2/doorControlPart/unlockedDoor AT 802 : BOOL := false;
    car2/doorL2/doorControlPart/openingRequest AT 803 : BOOL := false;
    car2/doorL2/doorControlPart/doorOpeningCmd AT 804 : BOOL := false;
    car2/doorL2/doorControlPart/doorClosingCmd AT 805 : BOOL := false;
    car2/doorL2/doorControlPart/doorLockingCmd AT 797 : BOOL := false;
    car2/doorL2/doorControlPart/doorUnlockingCmd AT 798 : BOOL := false;
    car2/doorL2/doorControlPart/closedDoorState AT 56 : BOOL := false;
    car2/doorL2/doorControlPart/openedDoorState AT 55 : BOOL := false;
    car2/doorL2/doorControlPart/faultState AT 539 : DINT := 0;
    car2/doorL2/doorControlPart/_X_10 AT 817 : BOOL := true;
    car2/doorL2/doorControlPart/_X_11 AT 818 : BOOL := false;
    car2/doorL2/doorControlPart/_X_12 AT 819 : BOOL := false;
    car2/doorL2/doorControlPart/_X_13 AT 820 : BOOL := false;
    car2/doorL2/doorControlPart/_X_14 AT 821 : BOOL := false;
    car2/doorL2/doorControlPart/_X_15 AT 822 : BOOL := false;
    car2/doorL2/doorControlPart/_X_16 AT 823 : BOOL := false;
    car2/doorL2/door/compressedAir AT 85 : REAL := 200.0;
    car2/doorL2/door/cmdSupply AT 730 : BOOL := true;
    car2/doorL2/door/sensorSupply AT 729 : BOOL := true;
    car2/doorL2/door/openDoorCmd AT 804 : BOOL := false;
    car2/doorL2/door/closeDoorCmd AT 805 : BOOL := false;
    car2/doorL2/door/lockActive AT 806 : BOOL := false;
    car2/doorL2/door/doorOpened AT 799 : BOOL := false;
    car2/doorL2/door/doorClosed AT 800 : BOOL := false;
    car2/doorL2/door/increment AT 91 : REAL := 0.0;
    car2/doorL2/door/openDoor AT 830 : BOOL := false;
    car2/doorL2/door/closeDoor AT 831 : BOOL := false;
    car2/doorL2/door/doorPosition AT 92 : REAL := 0.0;
    car2/doorL2/door/length AT 93 : REAL := 1000.0;
    car2/doorL2/door/doorClosedSensorLogic AT 832 : BOOL := true;
    car2/doorL2/door/doorOpenedSensorLogic AT 833 : BOOL := true;
    car2/doorL2/door/d_locking AT 834 : BOOL := false;
    car2/doorL2/door/v_d_locking AT 94 : REAL := 50.0;
    car2/doorL2/door/d_doorClosedSensor AT 835 : BOOL := false;
    car2/doorL2/door/v_d_doorClosedSensor AT 836 : BOOL := false;
    car2/doorL2/door/d_doorOpenedSensor AT 837 : BOOL := false;
    car2/doorL2/door/v_d_doorOpenedSensor AT 838 : BOOL := false;
    car2/doorL3/compressedAir AT 84 : REAL := 200.0;
    car2/doorL3/cmdSupply AT 728 : BOOL := true;
    car2/doorL3/sensorSupply AT 727 : BOOL := true;
    car2/doorL3/enableOpening AT 733 : BOOL := false;
    car2/doorL3/enableClosing AT 734 : BOOL := false;
    car2/doorL3/closedDoorState AT 54 : BOOL := false;
    car2/doorL3/openedDoorState AT 53 : BOOL := false;
    car2/doorL3/faultState AT 538 : DINT := 0;
    car2/doorL3/doorPB/doorPB AT 845 : BOOL := false;
    car2/doorL3/doorPB/button AT 849 : BOOL := false;
    car2/doorL3/doorPB/_X_10 AT 850 : BOOL := true;
    car2/doorL3/doorPB/_X_11 AT 851 : BOOL := false;
    car2/doorL3/doorPB/_X_12 AT 852 : BOOL := false;
    car2/doorL3/doorLocking/lockingCmd AT 839 : BOOL := false;
    car2/doorL3/doorLocking/unlockingCmd AT 840 : BOOL := false;
    car2/doorL3/doorLocking/doorLocked AT 843 : BOOL := false;
    car2/doorL3/doorLocking/doorUnlocked AT 844 : BOOL := false;
    car2/doorL3/doorLocking/lockActive AT 848 : BOOL := false;
    car2/doorL3/doorLocking/i_rs1 AT 632 : DINT := 0;
    car2/doorL3/doorLocking/d_unlockedSensor AT 854 : BOOL := false;
    car2/doorL3/doorLocking/v_d_unlockedSensor AT 855 : BOOL := false;
    car2/doorL3/doorLocking/d_lockedSensor AT 856 : BOOL := false;
    car2/doorL3/doorLocking/v_d_lockedSensor AT 857 : BOOL := false;
    car2/doorL3/doorControlPart/enableOpening AT 733 : BOOL := false;
    car2/doorL3/doorControlPart/enableClosing AT 734 : BOOL := false;
    car2/doorL3/doorControlPart/openedDoor AT 841 : BOOL := false;
    car2/doorL3/doorControlPart/closedDoor AT 842 : BOOL := false;
    car2/doorL3/doorControlPart/lockedDoor AT 843 : BOOL := false;
    car2/doorL3/doorControlPart/unlockedDoor AT 844 : BOOL := false;
    car2/doorL3/doorControlPart/openingRequest AT 845 : BOOL := false;
    car2/doorL3/doorControlPart/doorOpeningCmd AT 846 : BOOL := false;
    car2/doorL3/doorControlPart/doorClosingCmd AT 847 : BOOL := false;
    car2/doorL3/doorControlPart/doorLockingCmd AT 839 : BOOL := false;
    car2/doorL3/doorControlPart/doorUnlockingCmd AT 840 : BOOL := false;
    car2/doorL3/doorControlPart/closedDoorState AT 54 : BOOL := false;
    car2/doorL3/doorControlPart/openedDoorState AT 53 : BOOL := false;
    car2/doorL3/doorControlPart/faultState AT 538 : DINT := 0;
    car2/doorL3/doorControlPart/_X_10 AT 859 : BOOL := true;
    car2/doorL3/doorControlPart/_X_11 AT 860 : BOOL := false;
    car2/doorL3/doorControlPart/_X_12 AT 861 : BOOL := false;
    car2/doorL3/doorControlPart/_X_13 AT 862 : BOOL := false;
    car2/doorL3/doorControlPart/_X_14 AT 863 : BOOL := false;
    car2/doorL3/doorControlPart/_X_15 AT 864 : BOOL := false;
    car2/doorL3/doorControlPart/_X_16 AT 865 : BOOL := false;
    car2/doorL3/door/compressedAir AT 84 : REAL := 200.0;
    car2/doorL3/door/cmdSupply AT 728 : BOOL := true;
    car2/doorL3/door/sensorSupply AT 727 : BOOL := true;
    car2/doorL3/door/openDoorCmd AT 846 : BOOL := false;
    car2/doorL3/door/closeDoorCmd AT 847 : BOOL := false;
    car2/doorL3/door/lockActive AT 848 : BOOL := false;
    car2/doorL3/door/doorOpened AT 841 : BOOL := false;
    car2/doorL3/door/doorClosed AT 842 : BOOL := false;
    car2/doorL3/door/increment AT 95 : REAL := 0.0;
    car2/doorL3/door/openDoor AT 872 : BOOL := false;
    car2/doorL3/door/closeDoor AT 873 : BOOL := false;
    car2/doorL3/door/doorPosition AT 96 : REAL := 0.0;
    car2/doorL3/door/length AT 97 : REAL := 1000.0;
    car2/doorL3/door/doorClosedSensorLogic AT 874 : BOOL := true;
    car2/doorL3/door/doorOpenedSensorLogic AT 875 : BOOL := true;
    car2/doorL3/door/d_locking AT 876 : BOOL := false;
    car2/doorL3/door/v_d_locking AT 98 : REAL := 50.0;
    car2/doorL3/door/d_doorClosedSensor AT 877 : BOOL := false;
    car2/doorL3/door/v_d_doorClosedSensor AT 878 : BOOL := false;
    car2/doorL3/door/d_doorOpenedSensor AT 879 : BOOL := false;
    car2/doorL3/door/v_d_doorOpenedSensor AT 880 : BOOL := false;
    car2/doorR1/compressedAir AT 83 : REAL := 200.0;
    car2/doorR1/cmdSupply AT 726 : BOOL := true;
    car2/doorR1/sensorSupply AT 725 : BOOL := true;
    car2/doorR1/enableOpening AT 735 : BOOL := false;
    car2/doorR1/enableClosing AT 736 : BOOL := false;
    car2/doorR1/closedDoorState AT 52 : BOOL := false;
    car2/doorR1/openedDoorState AT 51 : BOOL := false;
    car2/doorR1/faultState AT 537 : DINT := 0;
    car2/doorR1/doorPB/doorPB AT 887 : BOOL := false;
    car2/doorR1/doorPB/button AT 891 : BOOL := false;
    car2/doorR1/doorPB/_X_10 AT 892 : BOOL := true;
    car2/doorR1/doorPB/_X_11 AT 893 : BOOL := false;
    car2/doorR1/doorPB/_X_12 AT 894 : BOOL := false;
    car2/doorR1/doorLocking/lockingCmd AT 881 : BOOL := false;
    car2/doorR1/doorLocking/unlockingCmd AT 882 : BOOL := false;
    car2/doorR1/doorLocking/doorLocked AT 885 : BOOL := false;
    car2/doorR1/doorLocking/doorUnlocked AT 886 : BOOL := false;
    car2/doorR1/doorLocking/lockActive AT 890 : BOOL := false;
    car2/doorR1/doorLocking/i_rs1 AT 635 : DINT := 0;
    car2/doorR1/doorLocking/d_unlockedSensor AT 896 : BOOL := false;
    car2/doorR1/doorLocking/v_d_unlockedSensor AT 897 : BOOL := false;
    car2/doorR1/doorLocking/d_lockedSensor AT 898 : BOOL := false;
    car2/doorR1/doorLocking/v_d_lockedSensor AT 899 : BOOL := false;
    car2/doorR1/doorControlPart/enableOpening AT 735 : BOOL := false;
    car2/doorR1/doorControlPart/enableClosing AT 736 : BOOL := false;
    car2/doorR1/doorControlPart/openedDoor AT 883 : BOOL := false;
    car2/doorR1/doorControlPart/closedDoor AT 884 : BOOL := false;
    car2/doorR1/doorControlPart/lockedDoor AT 885 : BOOL := false;
    car2/doorR1/doorControlPart/unlockedDoor AT 886 : BOOL := false;
    car2/doorR1/doorControlPart/openingRequest AT 887 : BOOL := false;
    car2/doorR1/doorControlPart/doorOpeningCmd AT 888 : BOOL := false;
    car2/doorR1/doorControlPart/doorClosingCmd AT 889 : BOOL := false;
    car2/doorR1/doorControlPart/doorLockingCmd AT 881 : BOOL := false;
    car2/doorR1/doorControlPart/doorUnlockingCmd AT 882 : BOOL := false;
    car2/doorR1/doorControlPart/closedDoorState AT 52 : BOOL := false;
    car2/doorR1/doorControlPart/openedDoorState AT 51 : BOOL := false;
    car2/doorR1/doorControlPart/faultState AT 537 : DINT := 0;
    car2/doorR1/doorControlPart/_X_10 AT 901 : BOOL := true;
    car2/doorR1/doorControlPart/_X_11 AT 902 : BOOL := false;
    car2/doorR1/doorControlPart/_X_12 AT 903 : BOOL := false;
    car2/doorR1/doorControlPart/_X_13 AT 904 : BOOL := false;
    car2/doorR1/doorControlPart/_X_14 AT 905 : BOOL := false;
    car2/doorR1/doorControlPart/_X_15 AT 906 : BOOL := false;
    car2/doorR1/doorControlPart/_X_16 AT 907 : BOOL := false;
    car2/doorR1/door/compressedAir AT 83 : REAL := 200.0;
    car2/doorR1/door/cmdSupply AT 726 : BOOL := true;
    car2/doorR1/door/sensorSupply AT 725 : BOOL := true;
    car2/doorR1/door/openDoorCmd AT 888 : BOOL := false;
    car2/doorR1/door/closeDoorCmd AT 889 : BOOL := false;
    car2/doorR1/door/lockActive AT 890 : BOOL := false;
    car2/doorR1/door/doorOpened AT 883 : BOOL := false;
    car2/doorR1/door/doorClosed AT 884 : BOOL := false;
    car2/doorR1/door/increment AT 99 : REAL := 0.0;
    car2/doorR1/door/openDoor AT 914 : BOOL := false;
    car2/doorR1/door/closeDoor AT 915 : BOOL := false;
    car2/doorR1/door/doorPosition AT 100 : REAL := 0.0;
    car2/doorR1/door/length AT 101 : REAL := 1000.0;
    car2/doorR1/door/doorClosedSensorLogic AT 916 : BOOL := true;
    car2/doorR1/door/doorOpenedSensorLogic AT 917 : BOOL := true;
    car2/doorR1/door/d_locking AT 918 : BOOL := false;
    car2/doorR1/door/v_d_locking AT 102 : REAL := 50.0;
    car2/doorR1/door/d_doorClosedSensor AT 919 : BOOL := false;
    car2/doorR1/door/v_d_doorClosedSensor AT 920 : BOOL := false;
    car2/doorR1/door/d_doorOpenedSensor AT 921 : BOOL := false;
    car2/doorR1/door/v_d_doorOpenedSensor AT 922 : BOOL := false;
    car2/doorR2/compressedAir AT 82 : REAL := 200.0;
    car2/doorR2/cmdSupply AT 724 : BOOL := true;
    car2/doorR2/sensorSupply AT 723 : BOOL := true;
    car2/doorR2/enableOpening AT 735 : BOOL := false;
    car2/doorR2/enableClosing AT 736 : BOOL := false;
    car2/doorR2/closedDoorState AT 50 : BOOL := false;
    car2/doorR2/openedDoorState AT 49 : BOOL := false;
    car2/doorR2/faultState AT 536 : DINT := 0;
    car2/doorR2/doorPB/doorPB AT 929 : BOOL := false;
    car2/doorR2/doorPB/button AT 933 : BOOL := false;
    car2/doorR2/doorPB/_X_10 AT 934 : BOOL := true;
    car2/doorR2/doorPB/_X_11 AT 935 : BOOL := false;
    car2/doorR2/doorPB/_X_12 AT 936 : BOOL := false;
    car2/doorR2/doorLocking/lockingCmd AT 923 : BOOL := false;
    car2/doorR2/doorLocking/unlockingCmd AT 924 : BOOL := false;
    car2/doorR2/doorLocking/doorLocked AT 927 : BOOL := false;
    car2/doorR2/doorLocking/doorUnlocked AT 928 : BOOL := false;
    car2/doorR2/doorLocking/lockActive AT 932 : BOOL := false;
    car2/doorR2/doorLocking/i_rs1 AT 638 : DINT := 0;
    car2/doorR2/doorLocking/d_unlockedSensor AT 938 : BOOL := false;
    car2/doorR2/doorLocking/v_d_unlockedSensor AT 939 : BOOL := false;
    car2/doorR2/doorLocking/d_lockedSensor AT 940 : BOOL := false;
    car2/doorR2/doorLocking/v_d_lockedSensor AT 941 : BOOL := false;
    car2/doorR2/doorControlPart/enableOpening AT 735 : BOOL := false;
    car2/doorR2/doorControlPart/enableClosing AT 736 : BOOL := false;
    car2/doorR2/doorControlPart/openedDoor AT 925 : BOOL := false;
    car2/doorR2/doorControlPart/closedDoor AT 926 : BOOL := false;
    car2/doorR2/doorControlPart/lockedDoor AT 927 : BOOL := false;
    car2/doorR2/doorControlPart/unlockedDoor AT 928 : BOOL := false;
    car2/doorR2/doorControlPart/openingRequest AT 929 : BOOL := false;
    car2/doorR2/doorControlPart/doorOpeningCmd AT 930 : BOOL := false;
    car2/doorR2/doorControlPart/doorClosingCmd AT 931 : BOOL := false;
    car2/doorR2/doorControlPart/doorLockingCmd AT 923 : BOOL := false;
    car2/doorR2/doorControlPart/doorUnlockingCmd AT 924 : BOOL := false;
    car2/doorR2/doorControlPart/closedDoorState AT 50 : BOOL := false;
    car2/doorR2/doorControlPart/openedDoorState AT 49 : BOOL := false;
    car2/doorR2/doorControlPart/faultState AT 536 : DINT := 0;
    car2/doorR2/doorControlPart/_X_10 AT 943 : BOOL := true;
    car2/doorR2/doorControlPart/_X_11 AT 944 : BOOL := false;
    car2/doorR2/doorControlPart/_X_12 AT 945 : BOOL := false;
    car2/doorR2/doorControlPart/_X_13 AT 946 : BOOL := false;
    car2/doorR2/doorControlPart/_X_14 AT 947 : BOOL := false;
    car2/doorR2/doorControlPart/_X_15 AT 948 : BOOL := false;
    car2/doorR2/doorControlPart/_X_16 AT 949 : BOOL := false;
    car2/doorR2/door/compressedAir AT 82 : REAL := 200.0;
    car2/doorR2/door/cmdSupply AT 724 : BOOL := true;
    car2/doorR2/door/sensorSupply AT 723 : BOOL := true;
    car2/doorR2/door/openDoorCmd AT 930 : BOOL := false;
    car2/doorR2/door/closeDoorCmd AT 931 : BOOL := false;
    car2/doorR2/door/lockActive AT 932 : BOOL := false;
    car2/doorR2/door/doorOpened AT 925 : BOOL := false;
    car2/doorR2/door/doorClosed AT 926 : BOOL := false;
    car2/doorR2/door/increment AT 103 : REAL := 0.0;
    car2/doorR2/door/openDoor AT 956 : BOOL := false;
    car2/doorR2/door/closeDoor AT 957 : BOOL := false;
    car2/doorR2/door/doorPosition AT 104 : REAL := 0.0;
    car2/doorR2/door/length AT 105 : REAL := 1000.0;
    car2/doorR2/door/doorClosedSensorLogic AT 958 : BOOL := true;
    car2/doorR2/door/doorOpenedSensorLogic AT 959 : BOOL := true;
    car2/doorR2/door/d_locking AT 960 : BOOL := false;
    car2/doorR2/door/v_d_locking AT 106 : REAL := 50.0;
    car2/doorR2/door/d_doorClosedSensor AT 961 : BOOL := false;
    car2/doorR2/door/v_d_doorClosedSensor AT 962 : BOOL := false;
    car2/doorR2/door/d_doorOpenedSensor AT 963 : BOOL := false;
    car2/doorR2/door/v_d_doorOpenedSensor AT 964 : BOOL := false;
    car2/doorR3/compressedAir AT 81 : REAL := 200.0;
    car2/doorR3/cmdSupply AT 722 : BOOL := true;
    car2/doorR3/sensorSupply AT 721 : BOOL := true;
    car2/doorR3/enableOpening AT 735 : BOOL := false;
    car2/doorR3/enableClosing AT 736 : BOOL := false;
    car2/doorR3/closedDoorState AT 48 : BOOL := false;
    car2/doorR3/openedDoorState AT 47 : BOOL := false;
    car2/doorR3/faultState AT 535 : DINT := 0;
    car2/doorR3/doorPB/doorPB AT 971 : BOOL := false;
    car2/doorR3/doorPB/button AT 975 : BOOL := false;
    car2/doorR3/doorPB/_X_10 AT 976 : BOOL := true;
    car2/doorR3/doorPB/_X_11 AT 977 : BOOL := false;
    car2/doorR3/doorPB/_X_12 AT 978 : BOOL := false;
    car2/doorR3/doorLocking/lockingCmd AT 965 : BOOL := false;
    car2/doorR3/doorLocking/unlockingCmd AT 966 : BOOL := false;
    car2/doorR3/doorLocking/doorLocked AT 969 : BOOL := false;
    car2/doorR3/doorLocking/doorUnlocked AT 970 : BOOL := false;
    car2/doorR3/doorLocking/lockActive AT 974 : BOOL := false;
    car2/doorR3/doorLocking/i_rs1 AT 641 : DINT := 0;
    car2/doorR3/doorLocking/d_unlockedSensor AT 980 : BOOL := false;
    car2/doorR3/doorLocking/v_d_unlockedSensor AT 981 : BOOL := false;
    car2/doorR3/doorLocking/d_lockedSensor AT 982 : BOOL := false;
    car2/doorR3/doorLocking/v_d_lockedSensor AT 983 : BOOL := false;
    car2/doorR3/doorControlPart/enableOpening AT 735 : BOOL := false;
    car2/doorR3/doorControlPart/enableClosing AT 736 : BOOL := false;
    car2/doorR3/doorControlPart/openedDoor AT 967 : BOOL := false;
    car2/doorR3/doorControlPart/closedDoor AT 968 : BOOL := false;
    car2/doorR3/doorControlPart/lockedDoor AT 969 : BOOL := false;
    car2/doorR3/doorControlPart/unlockedDoor AT 970 : BOOL := false;
    car2/doorR3/doorControlPart/openingRequest AT 971 : BOOL := false;
    car2/doorR3/doorControlPart/doorOpeningCmd AT 972 : BOOL := false;
    car2/doorR3/doorControlPart/doorClosingCmd AT 973 : BOOL := false;
    car2/doorR3/doorControlPart/doorLockingCmd AT 965 : BOOL := false;
    car2/doorR3/doorControlPart/doorUnlockingCmd AT 966 : BOOL := false;
    car2/doorR3/doorControlPart/closedDoorState AT 48 : BOOL := false;
    car2/doorR3/doorControlPart/openedDoorState AT 47 : BOOL := false;
    car2/doorR3/doorControlPart/faultState AT 535 : DINT := 0;
    car2/doorR3/doorControlPart/_X_10 AT 985 : BOOL := true;
    car2/doorR3/doorControlPart/_X_11 AT 986 : BOOL := false;
    car2/doorR3/doorControlPart/_X_12 AT 987 : BOOL := false;
    car2/doorR3/doorControlPart/_X_13 AT 988 : BOOL := false;
    car2/doorR3/doorControlPart/_X_14 AT 989 : BOOL := false;
    car2/doorR3/doorControlPart/_X_15 AT 990 : BOOL := false;
    car2/doorR3/doorControlPart/_X_16 AT 991 : BOOL := false;
    car2/doorR3/door/compressedAir AT 81 : REAL := 200.0;
    car2/doorR3/door/cmdSupply AT 722 : BOOL := true;
    car2/doorR3/door/sensorSupply AT 721 : BOOL := true;
    car2/doorR3/door/openDoorCmd AT 972 : BOOL := false;
    car2/doorR3/door/closeDoorCmd AT 973 : BOOL := false;
    car2/doorR3/door/lockActive AT 974 : BOOL := false;
    car2/doorR3/door/doorOpened AT 967 : BOOL := false;
    car2/doorR3/door/doorClosed AT 968 : BOOL := false;
    car2/doorR3/door/increment AT 107 : REAL := 0.0;
    car2/doorR3/door/openDoor AT 998 : BOOL := false;
    car2/doorR3/door/closeDoor AT 999 : BOOL := false;
    car2/doorR3/door/doorPosition AT 108 : REAL := 0.0;
    car2/doorR3/door/length AT 109 : REAL := 1000.0;
    car2/doorR3/door/doorClosedSensorLogic AT 1000 : BOOL := true;
    car2/doorR3/door/doorOpenedSensorLogic AT 1001 : BOOL := true;
    car2/doorR3/door/d_locking AT 1002 : BOOL := false;
    car2/doorR3/door/v_d_locking AT 110 : REAL := 50.0;
    car2/doorR3/door/d_doorClosedSensor AT 1003 : BOOL := false;
    car2/doorR3/door/v_d_doorClosedSensor AT 1004 : BOOL := false;
    car2/doorR3/door/d_doorOpenedSensor AT 1005 : BOOL := false;
    car2/doorR3/door/v_d_doorOpenedSensor AT 1006 : BOOL := false;
    car3/AuthorizationClosingLeftC1 AT 101 : BOOL := false;
    car3/AuthorizationOpeningRightC1 AT 102 : BOOL := false;
    car3/AuthorizationClosingRightC1 AT 103 : BOOL := false;
    car3/AuthorizationOpeningLeftC1 AT 104 : BOOL := false;
    car3/AuthorizationClosingLeftC2 AT 105 : BOOL := false;
    car3/AuthorizationOpeningRightC2 AT 106 : BOOL := false;
    car3/AuthorizationClosingRightC2 AT 107 : BOOL := false;
    car3/AuthorizationOpeningLeftC2 AT 108 : BOOL := false;
    car3/doorL1Closed AT 40 : BOOL := false;
    car3/doorL1Opened AT 39 : BOOL := false;
    car3/doorL1Fault AT 534 : DINT := 0;
    car3/doorL2Closed AT 38 : BOOL := false;
    car3/doorL2Opened AT 37 : BOOL := false;
    car3/doorL2Fault AT 533 : DINT := 0;
    car3/doorL3Closed AT 36 : BOOL := false;
    car3/doorL3Opened AT 35 : BOOL := false;
    car3/doorL3Fault AT 532 : DINT := 0;
    car3/doorR1Closed AT 34 : BOOL := false;
    car3/doorR1Opened AT 33 : BOOL := false;
    car3/doorR1Fault AT 531 : DINT := 0;
    car3/doorR2Closed AT 32 : BOOL := false;
    car3/doorR2Opened AT 31 : BOOL := false;
    car3/doorR2Fault AT 530 : DINT := 0;
    car3/doorR3Closed AT 30 : BOOL := false;
    car3/doorR3Opened AT 29 : BOOL := false;
    car3/doorR3Fault AT 529 : DINT := 0;
    car3/AlarmD1L AT 28 : BOOL := false;
    car3/AlarmD2L AT 27 : BOOL := false;
    car3/AlarmD3L AT 26 : BOOL := false;
    car3/AlarmD1R AT 25 : BOOL := false;
    car3/AlarmD2R AT 24 : BOOL := false;
    car3/AlarmD3R AT 23 : BOOL := false;
    car3/authorizations/AuthorizationClosingLeftC1 AT 101 : BOOL := false;
    car3/authorizations/AuthorizationOpeningRightC1 AT 102 : BOOL := false;
    car3/authorizations/AuthorizationClosingRightC1 AT 103 : BOOL := false;
    car3/authorizations/AuthorizationOpeningLeftC1 AT 104 : BOOL := false;
    car3/authorizations/AuthorizationClosingLeftC2 AT 105 : BOOL := false;
    car3/authorizations/AuthorizationOpeningRightC2 AT 106 : BOOL := false;
    car3/authorizations/AuthorizationClosingRightC2 AT 107 : BOOL := false;
    car3/authorizations/AuthorizationOpeningLeftC2 AT 108 : BOOL := false;
    car3/authorizations/AuthorizationOpeningLeft AT 1019 : BOOL := false;
    car3/authorizations/AuthorizationClosingLeft AT 1020 : BOOL := false;
    car3/authorizations/AuthorizationOpeningRight AT 1021 : BOOL := false;
    car3/authorizations/AuthorizationClosingRight AT 1022 : BOOL := false;
    car3/alarms/AlarmD1L AT 28 : BOOL := false;
    car3/alarms/AlarmD2L AT 27 : BOOL := false;
    car3/alarms/AlarmD3L AT 26 : BOOL := false;
    car3/alarms/AlarmD1R AT 25 : BOOL := false;
    car3/alarms/AlarmD2R AT 24 : BOOL := false;
    car3/alarms/AlarmD3R AT 23 : BOOL := false;
    car3/alarms/AlarmD1L/enableAlarm AT 1034 : BOOL := false;
    car3/alarms/AlarmD1L/resetKey AT 1033 : BOOL := false;
    car3/alarms/AlarmD1L/alarm AT 28 : BOOL := false;
    car3/alarms/AlarmD1L/i_rs1 AT 643 : DINT := 0;
    car3/alarms/AlarmD2L/enableAlarm AT 1032 : BOOL := false;
    car3/alarms/AlarmD2L/resetKey AT 1031 : BOOL := false;
    car3/alarms/AlarmD2L/alarm AT 27 : BOOL := false;
    car3/alarms/AlarmD2L/i_rs1 AT 645 : DINT := 0;
    car3/alarms/AlarmD3L/enableAlarm AT 1030 : BOOL := false;
    car3/alarms/AlarmD3L/resetKey AT 1029 : BOOL := false;
    car3/alarms/AlarmD3L/alarm AT 26 : BOOL := false;
    car3/alarms/AlarmD3L/i_rs1 AT 647 : DINT := 0;
    car3/alarms/AlarmD1R/enableAlarm AT 1028 : BOOL := false;
    car3/alarms/AlarmD1R/resetKey AT 1027 : BOOL := false;
    car3/alarms/AlarmD1R/alarm AT 25 : BOOL := false;
    car3/alarms/AlarmD1R/i_rs1 AT 649 : DINT := 0;
    car3/alarms/AlarmD2R/enableAlarm AT 1026 : BOOL := false;
    car3/alarms/AlarmD2R/resetKey AT 1025 : BOOL := false;
    car3/alarms/AlarmD2R/alarm AT 24 : BOOL := false;
    car3/alarms/AlarmD2R/i_rs1 AT 651 : DINT := 0;
    car3/alarms/AlarmD3R/enableAlarm AT 1024 : BOOL := false;
    car3/alarms/AlarmD3R/resetKey AT 1023 : BOOL := false;
    car3/alarms/AlarmD3R/alarm AT 23 : BOOL := false;
    car3/alarms/AlarmD3R/i_rs1 AT 653 : DINT := 0;
    car3/doorL1/compressedAir AT 116 : REAL := 200.0;
    car3/doorL1/cmdSupply AT 1018 : BOOL := true;
    car3/doorL1/sensorSupply AT 1017 : BOOL := true;
    car3/doorL1/enableOpening AT 1019 : BOOL := false;
    car3/doorL1/enableClosing AT 1020 : BOOL := false;
    car3/doorL1/closedDoorState AT 40 : BOOL := false;
    car3/doorL1/openedDoorState AT 39 : BOOL := false;
    car3/doorL1/faultState AT 534 : DINT := 0;
    car3/doorL1/doorPB/doorPB AT 1047 : BOOL := false;
    car3/doorL1/doorPB/button AT 1051 : BOOL := false;
    car3/doorL1/doorPB/_X_10 AT 1052 : BOOL := true;
    car3/doorL1/doorPB/_X_11 AT 1053 : BOOL := false;
    car3/doorL1/doorPB/_X_12 AT 1054 : BOOL := false;
    car3/doorL1/doorLocking/lockingCmd AT 1041 : BOOL := false;
    car3/doorL1/doorLocking/unlockingCmd AT 1042 : BOOL := false;
    car3/doorL1/doorLocking/doorLocked AT 1045 : BOOL := false;
    car3/doorL1/doorLocking/doorUnlocked AT 1046 : BOOL := false;
    car3/doorL1/doorLocking/lockActive AT 1050 : BOOL := false;
    car3/doorL1/doorLocking/i_rs1 AT 656 : DINT := 0;
    car3/doorL1/doorLocking/d_unlockedSensor AT 1056 : BOOL := false;
    car3/doorL1/doorLocking/v_d_unlockedSensor AT 1057 : BOOL := false;
    car3/doorL1/doorLocking/d_lockedSensor AT 1058 : BOOL := false;
    car3/doorL1/doorLocking/v_d_lockedSensor AT 1059 : BOOL := false;
    car3/doorL1/doorControlPart/enableOpening AT 1019 : BOOL := false;
    car3/doorL1/doorControlPart/enableClosing AT 1020 : BOOL := false;
    car3/doorL1/doorControlPart/openedDoor AT 1043 : BOOL := false;
    car3/doorL1/doorControlPart/closedDoor AT 1044 : BOOL := false;
    car3/doorL1/doorControlPart/lockedDoor AT 1045 : BOOL := false;
    car3/doorL1/doorControlPart/unlockedDoor AT 1046 : BOOL := false;
    car3/doorL1/doorControlPart/openingRequest AT 1047 : BOOL := false;
    car3/doorL1/doorControlPart/doorOpeningCmd AT 1048 : BOOL := false;
    car3/doorL1/doorControlPart/doorClosingCmd AT 1049 : BOOL := false;
    car3/doorL1/doorControlPart/doorLockingCmd AT 1041 : BOOL := false;
    car3/doorL1/doorControlPart/doorUnlockingCmd AT 1042 : BOOL := false;
    car3/doorL1/doorControlPart/closedDoorState AT 40 : BOOL := false;
    car3/doorL1/doorControlPart/openedDoorState AT 39 : BOOL := false;
    car3/doorL1/doorControlPart/faultState AT 534 : DINT := 0;
    car3/doorL1/doorControlPart/_X_10 AT 1061 : BOOL := true;
    car3/doorL1/doorControlPart/_X_11 AT 1062 : BOOL := false;
    car3/doorL1/doorControlPart/_X_12 AT 1063 : BOOL := false;
    car3/doorL1/doorControlPart/_X_13 AT 1064 : BOOL := false;
    car3/doorL1/doorControlPart/_X_14 AT 1065 : BOOL := false;
    car3/doorL1/doorControlPart/_X_15 AT 1066 : BOOL := false;
    car3/doorL1/doorControlPart/_X_16 AT 1067 : BOOL := false;
    car3/doorL1/door/compressedAir AT 116 : REAL := 200.0;
    car3/doorL1/door/cmdSupply AT 1018 : BOOL := true;
    car3/doorL1/door/sensorSupply AT 1017 : BOOL := true;
    car3/doorL1/door/openDoorCmd AT 1048 : BOOL := false;
    car3/doorL1/door/closeDoorCmd AT 1049 : BOOL := false;
    car3/doorL1/door/lockActive AT 1050 : BOOL := false;
    car3/doorL1/door/doorOpened AT 1043 : BOOL := false;
    car3/doorL1/door/doorClosed AT 1044 : BOOL := false;
    car3/doorL1/door/increment AT 117 : REAL := 0.0;
    car3/doorL1/door/openDoor AT 1074 : BOOL := false;
    car3/doorL1/door/closeDoor AT 1075 : BOOL := false;
    car3/doorL1/door/doorPosition AT 118 : REAL := 0.0;
    car3/doorL1/door/length AT 119 : REAL := 1000.0;
    car3/doorL1/door/doorClosedSensorLogic AT 1076 : BOOL := true;
    car3/doorL1/door/doorOpenedSensorLogic AT 1077 : BOOL := true;
    car3/doorL1/door/d_locking AT 1078 : BOOL := false;
    car3/doorL1/door/v_d_locking AT 120 : REAL := 50.0;
    car3/doorL1/door/d_doorClosedSensor AT 1079 : BOOL := false;
    car3/doorL1/door/v_d_doorClosedSensor AT 1080 : BOOL := false;
    car3/doorL1/door/d_doorOpenedSensor AT 1081 : BOOL := false;
    car3/doorL1/door/v_d_doorOpenedSensor AT 1082 : BOOL := false;
    car3/doorL2/compressedAir AT 115 : REAL := 200.0;
    car3/doorL2/cmdSupply AT 1016 : BOOL := true;
    car3/doorL2/sensorSupply AT 1015 : BOOL := true;
    car3/doorL2/enableOpening AT 1019 : BOOL := false;
    car3/doorL2/enableClosing AT 1020 : BOOL := false;
    car3/doorL2/closedDoorState AT 38 : BOOL := false;
    car3/doorL2/openedDoorState AT 37 : BOOL := false;
    car3/doorL2/faultState AT 533 : DINT := 0;
    car3/doorL2/doorPB/doorPB AT 1089 : BOOL := false;
    car3/doorL2/doorPB/button AT 1093 : BOOL := false;
    car3/doorL2/doorPB/_X_10 AT 1094 : BOOL := true;
    car3/doorL2/doorPB/_X_11 AT 1095 : BOOL := false;
    car3/doorL2/doorPB/_X_12 AT 1096 : BOOL := false;
    car3/doorL2/doorLocking/lockingCmd AT 1083 : BOOL := false;
    car3/doorL2/doorLocking/unlockingCmd AT 1084 : BOOL := false;
    car3/doorL2/doorLocking/doorLocked AT 1087 : BOOL := false;
    car3/doorL2/doorLocking/doorUnlocked AT 1088 : BOOL := false;
    car3/doorL2/doorLocking/lockActive AT 1092 : BOOL := false;
    car3/doorL2/doorLocking/i_rs1 AT 659 : DINT := 0;
    car3/doorL2/doorLocking/d_unlockedSensor AT 1098 : BOOL := false;
    car3/doorL2/doorLocking/v_d_unlockedSensor AT 1099 : BOOL := false;
    car3/doorL2/doorLocking/d_lockedSensor AT 1100 : BOOL := false;
    car3/doorL2/doorLocking/v_d_lockedSensor AT 1101 : BOOL := false;
    car3/doorL2/doorControlPart/enableOpening AT 1019 : BOOL := false;
    car3/doorL2/doorControlPart/enableClosing AT 1020 : BOOL := false;
